    |   movel([0.307212, -1.318657, -2.613011, -0.780720, 1.570796, 1.878009],accel_mss,speed_ms,0,blend_radius_m)
    |   movel([0.307312, -1.318721, -2.612972, -0.780696, 1.570796, 1.878109],accel_mss,speed_ms,0,blend_radius_m)
    |   movel([0.307553, -1.318455, -2.613136, -0.780797, 1.570796, 1.878349],accel_mss,speed_ms,0,blend_radius_m)
    |   movel([0.309131, -1.316503, -2.614344, -0.781542, 1.570796, 1.879927],accel_mss,speed_ms,0,blend_radius_m)
    |   movel([0.310529, -1.314958, -2.615295, -0.782136, 1.570796, 1.881325],accel_mss,speed_ms,0,blend_radius_m)
    |   movel([0.313319, -1.312233, -2.616967, -0.783190, 1.570796, 1.884115],accel_mss,speed_ms,0,blend_radius_m)
    |   movel([0.314719, -1.311087, -2.617666, -0.783636, 1.570796, 1.885515],accel_mss,speed_ms,0,blend_radius_m)
    |   movel([0.316170, -1.310050, -2.618298, -0.784041, 1.570796, 1.886966],accel_mss,speed_ms,0,blend_radius_m)
    |   movel([0.317768, -1.309055, -2.618903, -0.784431, 1.570796, 1.888565],accel_mss,speed_ms,0,blend_radius_m)
    |   movel([0.321234, -1.307125, -2.620073, -0.785192, 1.570796, 1.892031],accel_mss,speed_ms,0,blend_radius_m)
    |   movel([0.322560, -1.306227, -2.620615, -0.785547, 1.570796, 1.893356],accel_mss,speed_ms,0,blend_radius_m)
    |   movel([0.323660, -1.305298, -2.621175, -0.785916, 1.570796, 1.894456],accel_mss,speed_ms,0,blend_radius_m)
    |   movel([0.324594, -1.304294, -2.621779, -0.786316, 1.570796, 1.895391],accel_mss,speed_ms,0,blend_radius_m)
    |   movel([0.325732, -1.302493, -2.622860, -0.787037, 1.570796, 1.896528],accel_mss,speed_ms,0,blend_radius_m)
    |   movel([0.326232, -1.301501, -2.623453, -0.787435, 1.570796, 1.897028],accel_mss,speed_ms,0,blend_radius_m)
    |   movel([0.326144, -1.301362, -2.623536, -0.787491, 1.570796, 1.896941],accel_mss,speed_ms,0,blend_radius_m)
    |   movel([0.325589, -1.301882, -2.623225, -0.787282, 1.570796, 1.896385],accel_mss,speed_ms,0,blend_radius_m)
    |   movel([0.325038, -1.302447, -2.622887, -0.787055, 1.570796, 1.895835],accel_mss,speed_ms,0,blend_radius_m)
    |   movel([0.323893, -1.303624, -2.622182, -0.786584, 1.570796, 1.894689],accel_mss,speed_ms,0,blend_radius_m)
    |   speed_ms = 0.005
    |   movel([0.323893, -1.294431, -2.617839, -0.800119, 1.570796, 1.894689],accel_mss,speed_ms,0,blend_radius_m)
    |   speed_ms = 0.040
    |   movel([0.326258, -1.294277, -2.617930, -0.800182, 1.570796, 1.897054],accel_mss,speed_ms,0,blend_radius_m)
    |   speed_ms = 0.005
    |   movel([0.326258, -1.303470, -2.622274, -0.786645, 1.570796, 1.897054],accel_mss,speed_ms,0,blend_radius_m)
    |   speed_ms = 0.025
    |   movel([0.326747, -1.302560, -2.622819, -0.787009, 1.570796, 1.897543],accel_mss,speed_ms,0,blend_radius_m)
    |   movel([0.327247, -1.301359, -2.623537, -0.787492, 1.570796, 1.898043],accel_mss,speed_ms,0,blend_radius_m)
    |   movel([0.327645, -1.300186, -2.624237, -0.787966, 1.570796, 1.898441],accel_mss,speed_ms,0,blend_radius_m)
    |   movel([0.327795, -1.299396, -2.624707, -0.788286, 1.570796, 1.898591],accel_mss,speed_ms,0,blend_radius_m)
    |   movel([0.327707, -1.299045, -2.624916, -0.788428, 1.570796, 1.898503],accel_mss,speed_ms,0,blend_radius_m)
    |   movel([0.327425, -1.298928, -2.624985, -0.788475, 1.570796, 1.898222],accel_mss,speed_ms,0,blend_radius_m)
    |   movel([0.327033, -1.299087, -2.624891, -0.788411, 1.570796, 1.897830],accel_mss,speed_ms,0,blend_radius_m)
    |   movel([0.326013, -1.300232, -2.624210, -0.787947, 1.570796, 1.896809],accel_mss,speed_ms,0,blend_radius_m)
    |   movel([0.325507, -1.300775, -2.623886, -0.787728, 1.570796, 1.896303],accel_mss,speed_ms,0,blend_radius_m)
    |   movel([0.321787, -1.304518, -2.621645, -0.786227, 1.570796, 1.892583],accel_mss,speed_ms,0,blend_radius_m)
    |   movel([0.320328, -1.305732, -2.620914, -0.785744, 1.570796, 1.891125],accel_mss,speed_ms,0,blend_radius_m)
    |   movel([0.315897, -1.308955, -2.618964, -0.784470, 1.570796, 1.886693],accel_mss,speed_ms,0,blend_radius_m)
    |   movel([0.313137, -1.310933, -2.617760, -0.783696, 1.570796, 1.883934],accel_mss,speed_ms,0,blend_radius_m)
    |   movel([0.311061, -1.312571, -2.616760, -0.783058, 1.570796, 1.881857],accel_mss,speed_ms,0,blend_radius_m)
    |   movel([0.309487, -1.314003, -2.615882, -0.782504, 1.570796, 1.880283],accel_mss,speed_ms,0,blend_radius_m)
    |   movel([0.308299, -1.315334, -2.615064, -0.781991, 1.570796, 1.879095],accel_mss,speed_ms,0,blend_radius_m)
    |   movel([0.306934, -1.317318, -2.613840, -0.781231, 1.570796, 1.877730],accel_mss,speed_ms,0,blend_radius_m)
    |   movel([0.306002, -1.319214, -2.612666, -0.780509, 1.570796, 1.876798],accel_mss,speed_ms,0,blend_radius_m)
    |   movel([0.305550, -1.320906, -2.611614, -0.779869, 1.570796, 1.876346],accel_mss,speed_ms,0,blend_radius_m)
    |   movel([0.305606, -1.322295, -2.610747, -0.779347, 1.570796, 1.876402],accel_mss,speed_ms,0,blend_radius_m)
    |   movel([0.305810, -1.322929, -2.610351, -0.779109, 1.570796, 1.876606],accel_mss,speed_ms,0,blend_radius_m)
    |   movel([0.306043, -1.323253, -2.610148, -0.778988, 1.570796, 1.876840],accel_mss,speed_ms,0,blend_radius_m)
    |   movel([0.306324, -1.323321, -2.610106, -0.778962, 1.570796, 1.877120],accel_mss,speed_ms,0,blend_radius_m)
    |   movel([0.306667, -1.323175, -2.610197, -0.779017, 1.570796, 1.877463],accel_mss,speed_ms,0,blend_radius_m)
    |   movel([0.306853, -1.323006, -2.610303, -0.779080, 1.570796, 1.877649],accel_mss,speed_ms,0,blend_radius_m)
    |   movel([0.306996, -1.322598, -2.610558, -0.779233, 1.570796, 1.877793],accel_mss,speed_ms,0,blend_radius_m)
    |   movel([0.306995, -1.322152, -2.610837, -0.779400, 1.570796, 1.877792],accel_mss,speed_ms,0,blend_radius_m)
    |   movel([0.307215, -1.320929, -2.611600, -0.779861, 1.570796, 1.878011],accel_mss,speed_ms,0,blend_radius_m)
    |   movel([0.307915, -1.319503, -2.612487, -0.780400, 1.570796, 1.878712],accel_mss,speed_ms,0,blend_radius_m)
    |   movel([0.309145, -1.317798, -2.613544, -0.781048, 1.570796, 1.879941],accel_mss,speed_ms,0,blend_radius_m)
    |   movel([0.310979, -1.315725, -2.614823, -0.781841, 1.570796, 1.881775],accel_mss,speed_ms,0,blend_radius_m)
    |   movel([0.313038, -1.313657, -2.616095, -0.782638, 1.570796, 1.883835],accel_mss,speed_ms,0,blend_radius_m)
    |   movel([0.314866, -1.312075, -2.617063, -0.783251, 1.570796, 1.885662],accel_mss,speed_ms,0,blend_radius_m)
    |   movel([0.316790, -1.310710, -2.617896, -0.783783, 1.570796, 1.887586],accel_mss,speed_ms,0,blend_radius_m)
    |   movel([0.319152, -1.309304, -2.618752, -0.784333, 1.570796, 1.889949],accel_mss,speed_ms,0,blend_radius_m)
    |   movel([0.322628, -1.307240, -2.620003, -0.785146, 1.570796, 1.893424],accel_mss,speed_ms,0,blend_radius_m)
    |   movel([0.323637, -1.306466, -2.620471, -0.785452, 1.570796, 1.894434],accel_mss,speed_ms,0,blend_radius_m)
    |   movel([0.324629, -1.305529, -2.621036, -0.785824, 1.570796, 1.895425],accel_mss,speed_ms,0,blend_radius_m)
    |   movel([0.325525, -1.304506, -2.621652, -0.786231, 1.570796, 1.896322],accel_mss,speed_ms,0,blend_radius_m)
    |   movel([0.326258, -1.303470, -2.622274, -0.786645, 1.570796, 1.897054],accel_mss,speed_ms,0,blend_radius_m)
    |   movel([0.326747, -1.302560, -2.622819, -0.787009, 1.570796, 1.897543],accel_mss,speed_ms,0,blend_radius_m)
    |   movel([0.327247, -1.301359, -2.623537, -0.787492, 1.570796, 1.898043],accel_mss,speed_ms,0,blend_radius_m)
    |   movel([0.327406, -1.300891, -2.623817, -0.787681, 1.570796, 1.898202],accel_mss,speed_ms,0,blend_radius_m)
    |   speed_ms = 0.005
    |   movel([0.327406, -1.291683, -2.619461, -0.801245, 1.570796, 1.898202],accel_mss,speed_ms,0,blend_radius_m)
    |   speed_ms = 0.040
    |   movel([0.337782, -1.301882, -2.613390, -0.797116, 1.570796, 1.908579],accel_mss,speed_ms,0,blend_radius_m)
    |   speed_ms = 0.005
    |   movel([0.337782, -1.311032, -2.617700, -0.783657, 1.570796, 1.908579],accel_mss,speed_ms,0,blend_radius_m)
    |   speed_ms = 0.025
    |   movel([0.338243, -1.310133, -2.618248, -0.784008, 1.570796, 1.909039],accel_mss,speed_ms,0,blend_radius_m)
    |   movel([0.339898, -1.306587, -2.620397, -0.785404, 1.570796, 1.910694],accel_mss,speed_ms,0,blend_radius_m)
    |   movel([0.340033, -1.306182, -2.620642, -0.785565, 1.570796, 1.910829],accel_mss,speed_ms,0,blend_radius_m)
    |   movel([0.339919, -1.305852, -2.620841, -0.785696, 1.570796, 1.910716],accel_mss,speed_ms,0,blend_radius_m)
    |   movel([0.339552, -1.305923, -2.620798, -0.785668, 1.570796, 1.910349],accel_mss,speed_ms,0,blend_radius_m)
    |   movel([0.339171, -1.306264, -2.620593, -0.785533, 1.570796, 1.909967],accel_mss,speed_ms,0,blend_radius_m)
    |   movel([0.338711, -1.306998, -2.620149, -0.785242, 1.570796, 1.909508],accel_mss,speed_ms,0,blend_radius_m)
    |   movel([0.336280, -1.311905, -2.617167, -0.783317, 1.570796, 1.907076],accel_mss,speed_ms,0,blend_radius_m)
    |   movel([0.335256, -1.313851, -2.615976, -0.782563, 1.570796, 1.906053],accel_mss,speed_ms,0,blend_radius_m)
    |   movel([0.335041, -1.314109, -2.615817, -0.782463, 1.570796, 1.905837],accel_mss,speed_ms,0,blend_radius_m)
    |   movel([0.333925, -1.313709, -2.616063, -0.782617, 1.570796, 1.904721],accel_mss,speed_ms,0,blend_radius_m)
    |   movel([0.333466, -1.313809, -2.616001, -0.782579, 1.570796, 1.904262],accel_mss,speed_ms,0,blend_radius_m)
    |   movel([0.332950, -1.314205, -2.615758, -0.782426, 1.570796, 1.903746],accel_mss,speed_ms,0,blend_radius_m)
    |   movel([0.332250, -1.315025, -2.615254, -0.782110, 1.570796, 1.903046],accel_mss,speed_ms,0,blend_radius_m)
    |   movel([0.330578, -1.316890, -2.614105, -0.781394, 1.570796, 1.901374],accel_mss,speed_ms,0,blend_radius_m)
    |   movel([0.329691, -1.317759, -2.613568, -0.781062, 1.570796, 1.900487],accel_mss,speed_ms,0,blend_radius_m)
    |   movel([0.329694, -1.317312, -2.613844, -0.781233, 1.570796, 1.900490],accel_mss,speed_ms,0,blend_radius_m)
    |   movel([0.329719, -1.317037, -2.614014, -0.781338, 1.570796, 1.900515],accel_mss,speed_ms,0,blend_radius_m)
    |   movel([0.330422, -1.313511, -2.616184, -0.782694, 1.570796, 1.901218],accel_mss,speed_ms,0,blend_radius_m)
    |   movel([0.330386, -1.313253, -2.616342, -0.782794, 1.570796, 1.901182],accel_mss,speed_ms,0,blend_radius_m)
    |   movel([0.330238, -1.313153, -2.616403, -0.782833, 1.570796, 1.901034],accel_mss,speed_ms,0,blend_radius_m)
    |   movel([0.330096, -1.313161, -2.616398, -0.782829, 1.570796, 1.900892],accel_mss,speed_ms,0,blend_radius_m)
    |   movel([0.329664, -1.313389, -2.616259, -0.782741, 1.570796, 1.900460],accel_mss,speed_ms,0,blend_radius_m)
    |   movel([0.329304, -1.314002, -2.615883, -0.782504, 1.570796, 1.900100],accel_mss,speed_ms,0,blend_radius_m)
    |   movel([0.328587, -1.317415, -2.613780, -0.781194, 1.570796, 1.899383],accel_mss,speed_ms,0,blend_radius_m)
    |   movel([0.328597, -1.318361, -2.613195, -0.780833, 1.570796, 1.899393],accel_mss,speed_ms,0,blend_radius_m)
    |   movel([0.328770, -1.318650, -2.613016, -0.780723, 1.570796, 1.899566],accel_mss,speed_ms,0,blend_radius_m)
    |   movel([0.329121, -1.318773, -2.612940, -0.780677, 1.570796, 1.899918],accel_mss,speed_ms,0,blend_radius_m)
    |   movel([0.329584, -1.318705, -2.612981, -0.780702, 1.570796, 1.900380],accel_mss,speed_ms,0,blend_radius_m)
    |   movel([0.330062, -1.318458, -2.613135, -0.780796, 1.570796, 1.900859],accel_mss,speed_ms,0,blend_radius_m)
    |   movel([0.330544, -1.318068, -2.613376, -0.780944, 1.570796, 1.901341],accel_mss,speed_ms,0,blend_radius_m)
    |   movel([0.331223, -1.317416, -2.613780, -0.781193, 1.570796, 1.902019],accel_mss,speed_ms,0,blend_radius_m)
    |   movel([0.333567, -1.314812, -2.615385, -0.782192, 1.570796, 1.904363],accel_mss,speed_ms,0,blend_radius_m)
    |   movel([0.334016, -1.315298, -2.615086, -0.782005, 1.570796, 1.904812],accel_mss,speed_ms,0,blend_radius_m)
    |   movel([0.334664, -1.315728, -2.614822, -0.781840, 1.570796, 1.905460],accel_mss,speed_ms,0,blend_radius_m)
    |   movel([0.334838, -1.315746, -2.614811, -0.781833, 1.570796, 1.905634],accel_mss,speed_ms,0,blend_radius_m)
    |   movel([0.335212, -1.315522, -2.614948, -0.781919, 1.570796, 1.906008],accel_mss,speed_ms,0,blend_radius_m)
    |   movel([0.335737, -1.314781, -2.615404, -0.782204, 1.570796, 1.906534],accel_mss,speed_ms,0,blend_radius_m)
    |   movel([0.337782, -1.311032, -2.617700, -0.783657, 1.570796, 1.908579],accel_mss,speed_ms,0,blend_radius_m)
    |   movel([0.338243, -1.310133, -2.618248, -0.784008, 1.570796, 1.909039],accel_mss,speed_ms,0,blend_radius_m)
    |   movel([0.339015, -1.308475, -2.619255, -0.784659, 1.570796, 1.909811],accel_mss,speed_ms,0,blend_radius_m)
    |   speed_ms = 0.005
    |   movel([0.339015, -1.299311, -2.614934, -0.798145, 1.570796, 1.909811],accel_mss,speed_ms,0,blend_radius_m)
    |   speed_ms = 0.040
    |   movel([0.312088, -1.325803, -2.598622, -0.787964, 1.570796, 1.882884],accel_mss,speed_ms,0,blend_radius_m)
    |   speed_ms = 0.005
    |   movel([0.312088, -1.334807, -2.602825, -0.774757, 1.570796, 1.882884],accel_mss,speed_ms,0,blend_radius_m)
    |   speed_ms = 0.025
    |   movel([0.308392, -1.337491, -2.601098, -0.773800, 1.570796, 1.879188],accel_mss,speed_ms,0,blend_radius_m)
    |   movel([0.307353, -1.338080, -2.600717, -0.773591, 1.570796, 1.878150],accel_mss,speed_ms,0,blend_radius_m)
    |   movel([0.306493, -1.338398, -2.600512, -0.773479, 1.570796, 1.877289],accel_mss,speed_ms,0,blend_radius_m)
    |   movel([0.305914, -1.338470, -2.600466, -0.773453, 1.570796, 1.876710],accel_mss,speed_ms,0,blend_radius_m)
    |   movel([0.305711, -1.338314, -2.600567, -0.773509, 1.570796, 1.876508],accel_mss,speed_ms,0,blend_radius_m)
    |   movel([0.305836, -1.337950, -2.600802, -0.773637, 1.570796, 1.876632],accel_mss,speed_ms,0,blend_radius_m)
    |   movel([0.308276, -1.335053, -2.602667, -0.774669, 1.570796, 1.879072],accel_mss,speed_ms,0,blend_radius_m)
    |   movel([0.309248, -1.333743, -2.603507, -0.775139, 1.570796, 1.880044],accel_mss,speed_ms,0,blend_radius_m)
    |   movel([0.310608, -1.331652, -2.604842, -0.775894, 1.570796, 1.881405],accel_mss,speed_ms,0,blend_radius_m)
    |   movel([0.310997, -1.330924, -2.605306, -0.776159, 1.570796, 1.881794],accel_mss,speed_ms,0,blend_radius_m)
    |   movel([0.312034, -1.328173, -2.607052, -0.777164, 1.570796, 1.882830],accel_mss,speed_ms,0,blend_radius_m)
    |   movel([0.312141, -1.327720, -2.607338, -0.777331, 1.570796, 1.882937],accel_mss,speed_ms,0,blend_radius_m)
    |   movel([0.311958, -1.327277, -2.607618, -0.777494, 1.570796, 1.882755],accel_mss,speed_ms,0,blend_radius_m)
    |   movel([0.311748, -1.327028, -2.607775, -0.777586, 1.570796, 1.882544],accel_mss,speed_ms,0,blend_radius_m)
    |   movel([0.311758, -1.326727, -2.607965, -0.777697, 1.570796, 1.882554],accel_mss,speed_ms,0,blend_radius_m)
    |   movel([0.311983, -1.326441, -2.608145, -0.777802, 1.570796, 1.882779],accel_mss,speed_ms,0,blend_radius_m)
    |   movel([0.312368, -1.326236, -2.608275, -0.777878, 1.570796, 1.883164],accel_mss,speed_ms,0,blend_radius_m)
    |   movel([0.312840, -1.326193, -2.608302, -0.777894, 1.570796, 1.883637],accel_mss,speed_ms,0,blend_radius_m)
    |   movel([0.313138, -1.326410, -2.608165, -0.777814, 1.570796, 1.883934],accel_mss,speed_ms,0,blend_radius_m)
    |   movel([0.313250, -1.326915, -2.607847, -0.777627, 1.570796, 1.884046],accel_mss,speed_ms,0,blend_radius_m)
    |   movel([0.313171, -1.327736, -2.607328, -0.777325, 1.570796, 1.883967],accel_mss,speed_ms,0,blend_radius_m)
    |   movel([0.312702, -1.329366, -2.606296, -0.776727, 1.570796, 1.883499],accel_mss,speed_ms,0,blend_radius_m)
    |   movel([0.311799, -1.331308, -2.605062, -0.776019, 1.570796, 1.882595],accel_mss,speed_ms,0,blend_radius_m)
    |   movel([0.310569, -1.333362, -2.603751, -0.775276, 1.570796, 1.881366],accel_mss,speed_ms,0,blend_radius_m)
    |   movel([0.308247, -1.336526, -2.601720, -0.774143, 1.570796, 1.879043],accel_mss,speed_ms,0,blend_radius_m)
    |   movel([0.309250, -1.335888, -2.602131, -0.774370, 1.570796, 1.880046],accel_mss,speed_ms,0,blend_radius_m)
    |   movel([0.310249, -1.335148, -2.602606, -0.774635, 1.570796, 1.881045],accel_mss,speed_ms,0,blend_radius_m)
    |   movel([0.313227, -1.332919, -2.604034, -0.775436, 1.570796, 1.884024],accel_mss,speed_ms,0,blend_radius_m)
    |   movel([0.314209, -1.332259, -2.604455, -0.775674, 1.570796, 1.885005],accel_mss,speed_ms,0,blend_radius_m)
    |   movel([0.314787, -1.331983, -2.604632, -0.775775, 1.570796, 1.885583],accel_mss,speed_ms,0,blend_radius_m)
    |   movel([0.315091, -1.332027, -2.604603, -0.775758, 1.570796, 1.885887],accel_mss,speed_ms,0,blend_radius_m)
    |   movel([0.315060, -1.332306, -2.604426, -0.775658, 1.570796, 1.885856],accel_mss,speed_ms,0,blend_radius_m)
    |   movel([0.314691, -1.332734, -2.604152, -0.775503, 1.570796, 1.885488],accel_mss,speed_ms,0,blend_radius_m)
    |   movel([0.312088, -1.334807, -2.602825, -0.774757, 1.570796, 1.882884],accel_mss,speed_ms,0,blend_radius_m)
    |   movel([0.309627, -1.336591, -2.601678, -0.774120, 1.570796, 1.880423],accel_mss,speed_ms,0,blend_radius_m)
    |   speed_ms = 0.005
    |   movel([0.309627, -1.327599, -2.597483, -0.787307, 1.570796, 1.880423],accel_mss,speed_ms,0,blend_radius_m)
    |   speed_ms = 0.040
    |   movel([0.307273, -1.324388, -2.599517, -0.788484, 1.570796, 1.878069],accel_mss,speed_ms,0,blend_radius_m)
    |   speed_ms = 0.005
    |   movel([0.307273, -1.333401, -2.603726, -0.775262, 1.570796, 1.878069],accel_mss,speed_ms,0,blend_radius_m)
    |   speed_ms = 0.025
    |   movel([0.308595, -1.332314, -2.604420, -0.775655, 1.570796, 1.879391],accel_mss,speed_ms,0,blend_radius_m)
    |   movel([0.309287, -1.331629, -2.604857, -0.775903, 1.570796, 1.880084],accel_mss,speed_ms,0,blend_radius_m)
    |   movel([0.309505, -1.331215, -2.605121, -0.776053, 1.570796, 1.880302],accel_mss,speed_ms,0,blend_radius_m)
    |   movel([0.309377, -1.330977, -2.605272, -0.776139, 1.570796, 1.880173],accel_mss,speed_ms,0,blend_radius_m)
    |   movel([0.309182, -1.331020, -2.605245, -0.776124, 1.570796, 1.879979],accel_mss,speed_ms,0,blend_radius_m)
    |   movel([0.308663, -1.331351, -2.605035, -0.776004, 1.570796, 1.879459],accel_mss,speed_ms,0,blend_radius_m)
    |   movel([0.304437, -1.334482, -2.603033, -0.774873, 1.570796, 1.875234],accel_mss,speed_ms,0,blend_radius_m)
    |   movel([0.301937, -1.336094, -2.601998, -0.774297, 1.570796, 1.872734],accel_mss,speed_ms,0,blend_radius_m)
    |   movel([0.299591, -1.337354, -2.601187, -0.773849, 1.570796, 1.870388],accel_mss,speed_ms,0,blend_radius_m)
    |   movel([0.297404, -1.338260, -2.600601, -0.773528, 1.570796, 1.868201],accel_mss,speed_ms,0,blend_radius_m)
    |   movel([0.295735, -1.338801, -2.600251, -0.773336, 1.570796, 1.866531],accel_mss,speed_ms,0,blend_radius_m)
    |   movel([0.298270, -1.336381, -2.601813, -0.774195, 1.570796, 1.869067],accel_mss,speed_ms,0,blend_radius_m)
    |   movel([0.299778, -1.334767, -2.602851, -0.774771, 1.570796, 1.870574],accel_mss,speed_ms,0,blend_radius_m)
    |   movel([0.301019, -1.333262, -2.603815, -0.775312, 1.570796, 1.871816],accel_mss,speed_ms,0,blend_radius_m)
    |   movel([0.301505, -1.332372, -2.604383, -0.775634, 1.570796, 1.872302],accel_mss,speed_ms,0,blend_radius_m)
    |   movel([0.301499, -1.332129, -2.604538, -0.775721, 1.570796, 1.872295],accel_mss,speed_ms,0,blend_radius_m)
    |   movel([0.301389, -1.332106, -2.604553, -0.775730, 1.570796, 1.872185],accel_mss,speed_ms,0,blend_radius_m)
    |   movel([0.300923, -1.332271, -2.604448, -0.775670, 1.570796, 1.871719],accel_mss,speed_ms,0,blend_radius_m)
    |   movel([0.300572, -1.332571, -2.604256, -0.775562, 1.570796, 1.871369],accel_mss,speed_ms,0,blend_radius_m)
    |   movel([0.299480, -1.333796, -2.603473, -0.775120, 1.570796, 1.870276],accel_mss,speed_ms,0,blend_radius_m)
    |   movel([0.298256, -1.335199, -2.602573, -0.774617, 1.570796, 1.869053],accel_mss,speed_ms,0,blend_radius_m)
    |   movel([0.297100, -1.336370, -2.601820, -0.774198, 1.570796, 1.867896],accel_mss,speed_ms,0,blend_radius_m)
    |   movel([0.295923, -1.337399, -2.601157, -0.773833, 1.570796, 1.866720],accel_mss,speed_ms,0,blend_radius_m)
    |   movel([0.293513, -1.339225, -2.599977, -0.773187, 1.570796, 1.864309],accel_mss,speed_ms,0,blend_radius_m)
    |   movel([0.293230, -1.339512, -2.599791, -0.773086, 1.570796, 1.864027],accel_mss,speed_ms,0,blend_radius_m)
    |   movel([0.293138, -1.339896, -2.599542, -0.772951, 1.570796, 1.863934],accel_mss,speed_ms,0,blend_radius_m)
    |   movel([0.293264, -1.339985, -2.599484, -0.772920, 1.570796, 1.864061],accel_mss,speed_ms,0,blend_radius_m)
    |   movel([0.294226, -1.339955, -2.599504, -0.772930, 1.570796, 1.865022],accel_mss,speed_ms,0,blend_radius_m)
    |   movel([0.295597, -1.339742, -2.599642, -0.773005, 1.570796, 1.866393],accel_mss,speed_ms,0,blend_radius_m)
    |   movel([0.297004, -1.339349, -2.599897, -0.773143, 1.570796, 1.867801],accel_mss,speed_ms,0,blend_radius_m)
    |   movel([0.298619, -1.338737, -2.600293, -0.773359, 1.570796, 1.869415],accel_mss,speed_ms,0,blend_radius_m)
    |   movel([0.300228, -1.337994, -2.600773, -0.773622, 1.570796, 1.871025],accel_mss,speed_ms,0,blend_radius_m)
    |   movel([0.301988, -1.337043, -2.601387, -0.773959, 1.570796, 1.872784],accel_mss,speed_ms,0,blend_radius_m)
    |   movel([0.303714, -1.335978, -2.602073, -0.774338, 1.570796, 1.874511],accel_mss,speed_ms,0,blend_radius_m)
    |   movel([0.305518, -1.334733, -2.602872, -0.774783, 1.570796, 1.876314],accel_mss,speed_ms,0,blend_radius_m)
    |   movel([0.307273, -1.333401, -2.603726, -0.775262, 1.570796, 1.878069],accel_mss,speed_ms,0,blend_radius_m)
    |   movel([0.308595, -1.332314, -2.604420, -0.775655, 1.570796, 1.879391],accel_mss,speed_ms,0,blend_radius_m)
    |   movel([0.309287, -1.331629, -2.604857, -0.775903, 1.570796, 1.880084],accel_mss,speed_ms,0,blend_radius_m)
    |   movel([0.309446, -1.331328, -2.605049, -0.776012, 1.570796, 1.880242],accel_mss,speed_ms,0,blend_radius_m)
    |   speed_ms = 0.005
    |   movel([0.309446, -1.322303, -2.600830, -0.789256, 1.570796, 1.880242],accel_mss,speed_ms,0,blend_radius_m)
    |   speed_ms = 0.040
    |   movel([0.281169, -1.327397, -2.597611, -0.787380, 1.570796, 1.851966],accel_mss,speed_ms,0,blend_radius_m)
    |   speed_ms = 0.005
    |   movel([0.281169, -1.336390, -2.601807, -0.774191, 1.570796, 1.851966],accel_mss,speed_ms,0,blend_radius_m)
    |   speed_ms = 0.025
    |   movel([0.281589, -1.336173, -2.601948, -0.774269, 1.570796, 1.852385],accel_mss,speed_ms,0,blend_radius_m)
    |   movel([0.281862, -1.335916, -2.602113, -0.774361, 1.570796, 1.852658],accel_mss,speed_ms,0,blend_radius_m)
    |   movel([0.281947, -1.335663, -2.602275, -0.774451, 1.570796, 1.852743],accel_mss,speed_ms,0,blend_radius_m)
    |   movel([0.281691, -1.335396, -2.602447, -0.774546, 1.570796, 1.852488],accel_mss,speed_ms,0,blend_radius_m)
    |   movel([0.281436, -1.335403, -2.602442, -0.774543, 1.570796, 1.852232],accel_mss,speed_ms,0,blend_radius_m)
    |   movel([0.280018, -1.335751, -2.602219, -0.774419, 1.570796, 1.850815],accel_mss,speed_ms,0,blend_radius_m)
    |   movel([0.279438, -1.335889, -2.602130, -0.774370, 1.570796, 1.850234],accel_mss,speed_ms,0,blend_radius_m)
    |   movel([0.277464, -1.336169, -2.601950, -0.774270, 1.570796, 1.848260],accel_mss,speed_ms,0,blend_radius_m)
    |   movel([0.276225, -1.336162, -2.601954, -0.774273, 1.570796, 1.847021],accel_mss,speed_ms,0,blend_radius_m)
    |   movel([0.274250, -1.335940, -2.602097, -0.774352, 1.570796, 1.845046],accel_mss,speed_ms,0,blend_radius_m)
    |   movel([0.273688, -1.335778, -2.602201, -0.774410, 1.570796, 1.844484],accel_mss,speed_ms,0,blend_radius_m)
    |   movel([0.274932, -1.335215, -2.602563, -0.774611, 1.570796, 1.845728],accel_mss,speed_ms,0,blend_radius_m)
    |   movel([0.276555, -1.334383, -2.603097, -0.774909, 1.570796, 1.847351],accel_mss,speed_ms,0,blend_radius_m)
    |   movel([0.278096, -1.333386, -2.603736, -0.775268, 1.570796, 1.848892],accel_mss,speed_ms,0,blend_radius_m)
    |   movel([0.279291, -1.332432, -2.604345, -0.775612, 1.570796, 1.850087],accel_mss,speed_ms,0,blend_radius_m)
    |   movel([0.279536, -1.332138, -2.604533, -0.775718, 1.570796, 1.850333],accel_mss,speed_ms,0,blend_radius_m)
    |   movel([0.279647, -1.331822, -2.604734, -0.775833, 1.570796, 1.850443],accel_mss,speed_ms,0,blend_radius_m)
    |   movel([0.279578, -1.331667, -2.604833, -0.775889, 1.570796, 1.850375],accel_mss,speed_ms,0,blend_radius_m)
    |   movel([0.279357, -1.331607, -2.604871, -0.775911, 1.570796, 1.850153],accel_mss,speed_ms,0,blend_radius_m)
    |   movel([0.277761, -1.331783, -2.604759, -0.775847, 1.570796, 1.848557],accel_mss,speed_ms,0,blend_radius_m)
    |   movel([0.275731, -1.331936, -2.604661, -0.775791, 1.570796, 1.846527],accel_mss,speed_ms,0,blend_radius_m)
    |   movel([0.274030, -1.331774, -2.604765, -0.775850, 1.570796, 1.844826],accel_mss,speed_ms,0,blend_radius_m)
    |   movel([0.272602, -1.331281, -2.605079, -0.776029, 1.570796, 1.843398],accel_mss,speed_ms,0,blend_radius_m)
    |   movel([0.271400, -1.330446, -2.605610, -0.776333, 1.570796, 1.842196],accel_mss,speed_ms,0,blend_radius_m)
    |   movel([0.270719, -1.329821, -2.606007, -0.776561, 1.570796, 1.841515],accel_mss,speed_ms,0,blend_radius_m)
    |   movel([0.272339, -1.329417, -2.606263, -0.776708, 1.570796, 1.843135],accel_mss,speed_ms,0,blend_radius_m)
    |   movel([0.273542, -1.328831, -2.606635, -0.776923, 1.570796, 1.844338],accel_mss,speed_ms,0,blend_radius_m)
    |   movel([0.274574, -1.328160, -2.607060, -0.777169, 1.570796, 1.845371],accel_mss,speed_ms,0,blend_radius_m)
    |   movel([0.274821, -1.327919, -2.607213, -0.777258, 1.570796, 1.845617],accel_mss,speed_ms,0,blend_radius_m)
    |   movel([0.274963, -1.327481, -2.607489, -0.777419, 1.570796, 1.845759],accel_mss,speed_ms,0,blend_radius_m)
    |   movel([0.274856, -1.327336, -2.607581, -0.777472, 1.570796, 1.845652],accel_mss,speed_ms,0,blend_radius_m)
    |   movel([0.273461, -1.326733, -2.607961, -0.777695, 1.570796, 1.844257],accel_mss,speed_ms,0,blend_radius_m)
    |   movel([0.272555, -1.326179, -2.608311, -0.777900, 1.570796, 1.843351],accel_mss,speed_ms,0,blend_radius_m)
    |   movel([0.270971, -1.324730, -2.609222, -0.778437, 1.570796, 1.841768],accel_mss,speed_ms,0,blend_radius_m)
    |   movel([0.270367, -1.323880, -2.609756, -0.778754, 1.570796, 1.841164],accel_mss,speed_ms,0,blend_radius_m)
    |   movel([0.268936, -1.321297, -2.611370, -0.779722, 1.570796, 1.839732],accel_mss,speed_ms,0,blend_radius_m)
    |   movel([0.269008, -1.321099, -2.611494, -0.779796, 1.570796, 1.839804],accel_mss,speed_ms,0,blend_radius_m)
    |   movel([0.269540, -1.321127, -2.611476, -0.779786, 1.570796, 1.840337],accel_mss,speed_ms,0,blend_radius_m)
    |   movel([0.270152, -1.321157, -2.611457, -0.779774, 1.570796, 1.840948],accel_mss,speed_ms,0,blend_radius_m)
    |   movel([0.271202, -1.321024, -2.611540, -0.779824, 1.570796, 1.841998],accel_mss,speed_ms,0,blend_radius_m)
    |   movel([0.272261, -1.320821, -2.611667, -0.779901, 1.570796, 1.843057],accel_mss,speed_ms,0,blend_radius_m)
    |   movel([0.272824, -1.320593, -2.611808, -0.779987, 1.570796, 1.843620],accel_mss,speed_ms,0,blend_radius_m)
    |   movel([0.272987, -1.320485, -2.611876, -0.780028, 1.570796, 1.843784],accel_mss,speed_ms,0,blend_radius_m)
    |   movel([0.273301, -1.320135, -2.612094, -0.780160, 1.570796, 1.844098],accel_mss,speed_ms,0,blend_radius_m)
    |   movel([0.273295, -1.319996, -2.612180, -0.780213, 1.570796, 1.844091],accel_mss,speed_ms,0,blend_radius_m)
    |   movel([0.270912, -1.316196, -2.614533, -0.781660, 1.570796, 1.841709],accel_mss,speed_ms,0,blend_radius_m)
    |   movel([0.270432, -1.315413, -2.615015, -0.781960, 1.570796, 1.841229],accel_mss,speed_ms,0,blend_radius_m)
    |   movel([0.269305, -1.313068, -2.616456, -0.782866, 1.570796, 1.840101],accel_mss,speed_ms,0,blend_radius_m)
    |   movel([0.268936, -1.312131, -2.617029, -0.783229, 1.570796, 1.839732],accel_mss,speed_ms,0,blend_radius_m)
    |   movel([0.268935, -1.311909, -2.617165, -0.783315, 1.570796, 1.839731],accel_mss,speed_ms,0,blend_radius_m)
    |   movel([0.271324, -1.312552, -2.616771, -0.783066, 1.570796, 1.842120],accel_mss,speed_ms,0,blend_radius_m)
    |   movel([0.271647, -1.312532, -2.616784, -0.783073, 1.570796, 1.842444],accel_mss,speed_ms,0,blend_radius_m)
    |   movel([0.271996, -1.312357, -2.616890, -0.783141, 1.570796, 1.842792],accel_mss,speed_ms,0,blend_radius_m)
    |   movel([0.272209, -1.312110, -2.617042, -0.783237, 1.570796, 1.843005],accel_mss,speed_ms,0,blend_radius_m)
    |   movel([0.272228, -1.311863, -2.617193, -0.783333, 1.570796, 1.843025],accel_mss,speed_ms,0,blend_radius_m)
    |   movel([0.271712, -1.310973, -2.617736, -0.783680, 1.570796, 1.842508],accel_mss,speed_ms,0,blend_radius_m)
    |   movel([0.270908, -1.309420, -2.618681, -0.784288, 1.570796, 1.841704],accel_mss,speed_ms,0,blend_radius_m)
    |   movel([0.270396, -1.307212, -2.620020, -0.785157, 1.570796, 1.841192],accel_mss,speed_ms,0,blend_radius_m)
    |   movel([0.270182, -1.304482, -2.621666, -0.786241, 1.570796, 1.840978],accel_mss,speed_ms,0,blend_radius_m)
    |   movel([0.270293, -1.301324, -2.623559, -0.787507, 1.570796, 1.841089],accel_mss,speed_ms,0,blend_radius_m)
    |   movel([0.270506, -1.299002, -2.624941, -0.788445, 1.570796, 1.841302],accel_mss,speed_ms,0,blend_radius_m)
    |   movel([0.271637, -1.300175, -2.624244, -0.787970, 1.570796, 1.842433],accel_mss,speed_ms,0,blend_radius_m)
    |   movel([0.272159, -1.300765, -2.623892, -0.787732, 1.570796, 1.842955],accel_mss,speed_ms,0,blend_radius_m)
    |   movel([0.272907, -1.301368, -2.623532, -0.787489, 1.570796, 1.843704],accel_mss,speed_ms,0,blend_radius_m)
    |   movel([0.273169, -1.301398, -2.623514, -0.787477, 1.570796, 1.843965],accel_mss,speed_ms,0,blend_radius_m)
    |   movel([0.273762, -1.301145, -2.623666, -0.787579, 1.570796, 1.844558],accel_mss,speed_ms,0,blend_radius_m)
    |   movel([0.273821, -1.301011, -2.623745, -0.787633, 1.570796, 1.844618],accel_mss,speed_ms,0,blend_radius_m)
    |   movel([0.273864, -1.299446, -2.624678, -0.788265, 1.570796, 1.844661],accel_mss,speed_ms,0,blend_radius_m)
    |   movel([0.273850, -1.298479, -2.625252, -0.788658, 1.570796, 1.844647],accel_mss,speed_ms,0,blend_radius_m)
    |   movel([0.273970, -1.291208, -2.629533, -0.791648, 1.570796, 1.844767],accel_mss,speed_ms,0,blend_radius_m)
    |   movel([0.274176, -1.287340, -2.631783, -0.793266, 1.570796, 1.844973],accel_mss,speed_ms,0,blend_radius_m)
    |   movel([0.274427, -1.286894, -2.632041, -0.793453, 1.570796, 1.845223],accel_mss,speed_ms,0,blend_radius_m)
    |   movel([0.275681, -1.288748, -2.630966, -0.792674, 1.570796, 1.846477],accel_mss,speed_ms,0,blend_radius_m)
    |   movel([0.276045, -1.289112, -2.630755, -0.792522, 1.570796, 1.846841],accel_mss,speed_ms,0,blend_radius_m)
    |   movel([0.276374, -1.289162, -2.630726, -0.792501, 1.570796, 1.847170],accel_mss,speed_ms,0,blend_radius_m)
    |   movel([0.276720, -1.288968, -2.630839, -0.792582, 1.570796, 1.847517],accel_mss,speed_ms,0,blend_radius_m)
    |   movel([0.276872, -1.288749, -2.630966, -0.792674, 1.570796, 1.847668],accel_mss,speed_ms,0,blend_radius_m)
    |   movel([0.276936, -1.288488, -2.631118, -0.792784, 1.570796, 1.847732],accel_mss,speed_ms,0,blend_radius_m)
    |   movel([0.276818, -1.287496, -2.631693, -0.793200, 1.570796, 1.847614],accel_mss,speed_ms,0,blend_radius_m)
    |   movel([0.276600, -1.285984, -2.632568, -0.793838, 1.570796, 1.847396],accel_mss,speed_ms,0,blend_radius_m)
    |   movel([0.276603, -1.284773, -2.633266, -0.794350, 1.570796, 1.847399],accel_mss,speed_ms,0,blend_radius_m)
    |   movel([0.276842, -1.283399, -2.634056, -0.794934, 1.570796, 1.847638],accel_mss,speed_ms,0,blend_radius_m)
    |   movel([0.278133, -1.279062, -2.636535, -0.796793, 1.570796, 1.848929],accel_mss,speed_ms,0,blend_radius_m)
    |   movel([0.278449, -1.278207, -2.637020, -0.797161, 1.570796, 1.849246],accel_mss,speed_ms,0,blend_radius_m)
    |   movel([0.278845, -1.277612, -2.637358, -0.797419, 1.570796, 1.849641],accel_mss,speed_ms,0,blend_radius_m)
    |   movel([0.279260, -1.278513, -2.636846, -0.797029, 1.570796, 1.850056],accel_mss,speed_ms,0,blend_radius_m)
    |   movel([0.279418, -1.279098, -2.636514, -0.796777, 1.570796, 1.850215],accel_mss,speed_ms,0,blend_radius_m)
    |   movel([0.279740, -1.279576, -2.636242, -0.796571, 1.570796, 1.850536],accel_mss,speed_ms,0,blend_radius_m)
    |   movel([0.279962, -1.279602, -2.636227, -0.796560, 1.570796, 1.850758],accel_mss,speed_ms,0,blend_radius_m)
    |   movel([0.280323, -1.279456, -2.636311, -0.796623, 1.570796, 1.851120],accel_mss,speed_ms,0,blend_radius_m)
    |   movel([0.280542, -1.279207, -2.636452, -0.796730, 1.570796, 1.851338],accel_mss,speed_ms,0,blend_radius_m)
    |   movel([0.280712, -1.277787, -2.637259, -0.797343, 1.570796, 1.851509],accel_mss,speed_ms,0,blend_radius_m)
    |   movel([0.280895, -1.276342, -2.638077, -0.797970, 1.570796, 1.851691],accel_mss,speed_ms,0,blend_radius_m)
    |   movel([0.281383, -1.274385, -2.639181, -0.798823, 1.570796, 1.852179],accel_mss,speed_ms,0,blend_radius_m)
    |   movel([0.282040, -1.272367, -2.640314, -0.799708, 1.570796, 1.852836],accel_mss,speed_ms,0,blend_radius_m)
    |   movel([0.283334, -1.269598, -2.641862, -0.800930, 1.570796, 1.854130],accel_mss,speed_ms,0,blend_radius_m)
    |   movel([0.284030, -1.268377, -2.642540, -0.801471, 1.570796, 1.854826],accel_mss,speed_ms,0,blend_radius_m)
    |   movel([0.285181, -1.266600, -2.643526, -0.802263, 1.570796, 1.855978],accel_mss,speed_ms,0,blend_radius_m)
    |   movel([0.278484, -1.290136, -2.630158, -0.792094, 1.570796, 1.849281],accel_mss,speed_ms,0,blend_radius_m)
    |   movel([0.276921, -1.295658, -2.626921, -0.789810, 1.570796, 1.847717],accel_mss,speed_ms,0,blend_radius_m)
    |   movel([0.275389, -1.301455, -2.623480, -0.787454, 1.570796, 1.846185],accel_mss,speed_ms,0,blend_radius_m)
    |   movel([0.274554, -1.306620, -2.620377, -0.785391, 1.570796, 1.845351],accel_mss,speed_ms,0,blend_radius_m)
    |   movel([0.274120, -1.311508, -2.617409, -0.783471, 1.570796, 1.844916],accel_mss,speed_ms,0,blend_radius_m)
    |   movel([0.274094, -1.315860, -2.614740, -0.781789, 1.570796, 1.844890],accel_mss,speed_ms,0,blend_radius_m)
    |   movel([0.274490, -1.319404, -2.612548, -0.780437, 1.570796, 1.845286],accel_mss,speed_ms,0,blend_radius_m)
    |   movel([0.274833, -1.320766, -2.611701, -0.779922, 1.570796, 1.845630],accel_mss,speed_ms,0,blend_radius_m)
    |   movel([0.275323, -1.322040, -2.610907, -0.779442, 1.570796, 1.846119],accel_mss,speed_ms,0,blend_radius_m)
    |   movel([0.275945, -1.323183, -2.610192, -0.779014, 1.570796, 1.846741],accel_mss,speed_ms,0,blend_radius_m)
    |   movel([0.276713, -1.324213, -2.609547, -0.778630, 1.570796, 1.847509],accel_mss,speed_ms,0,blend_radius_m)
    |   movel([0.277660, -1.325170, -2.608946, -0.778273, 1.570796, 1.848457],accel_mss,speed_ms,0,blend_radius_m)
    |   movel([0.278736, -1.326004, -2.608421, -0.777964, 1.570796, 1.849532],accel_mss,speed_ms,0,blend_radius_m)
    |   movel([0.280052, -1.326810, -2.607913, -0.777666, 1.570796, 1.850848],accel_mss,speed_ms,0,blend_radius_m)
    |   movel([0.282073, -1.327768, -2.607308, -0.777313, 1.570796, 1.852870],accel_mss,speed_ms,0,blend_radius_m)
    |   movel([0.282343, -1.327826, -2.607271, -0.777292, 1.570796, 1.853139],accel_mss,speed_ms,0,blend_radius_m)
    |   movel([0.282844, -1.327570, -2.607433, -0.777386, 1.570796, 1.853640],accel_mss,speed_ms,0,blend_radius_m)
    |   movel([0.283094, -1.327338, -2.607579, -0.777471, 1.570796, 1.853890],accel_mss,speed_ms,0,blend_radius_m)
    |   movel([0.283122, -1.327095, -2.607733, -0.777561, 1.570796, 1.853918],accel_mss,speed_ms,0,blend_radius_m)
    |   movel([0.282896, -1.326892, -2.607861, -0.777636, 1.570796, 1.853692],accel_mss,speed_ms,0,blend_radius_m)
    |   movel([0.281185, -1.325946, -2.608457, -0.777986, 1.570796, 1.851981],accel_mss,speed_ms,0,blend_radius_m)
    |   movel([0.279868, -1.325215, -2.608917, -0.778257, 1.570796, 1.850665],accel_mss,speed_ms,0,blend_radius_m)
    |   movel([0.278657, -1.324324, -2.609477, -0.778588, 1.570796, 1.849453],accel_mss,speed_ms,0,blend_radius_m)
    |   movel([0.277641, -1.323357, -2.610083, -0.778949, 1.570796, 1.848437],accel_mss,speed_ms,0,blend_radius_m)
    |   movel([0.276926, -1.322389, -2.610688, -0.779311, 1.570796, 1.847722],accel_mss,speed_ms,0,blend_radius_m)
    |   movel([0.276395, -1.321223, -2.611416, -0.779750, 1.570796, 1.847191],accel_mss,speed_ms,0,blend_radius_m)
    |   movel([0.275478, -1.317626, -2.613650, -0.781113, 1.570796, 1.846274],accel_mss,speed_ms,0,blend_radius_m)
    |   movel([0.275265, -1.315892, -2.614720, -0.781776, 1.570796, 1.846061],accel_mss,speed_ms,0,blend_radius_m)
    |   movel([0.275198, -1.314070, -2.615841, -0.782478, 1.570796, 1.845995],accel_mss,speed_ms,0,blend_radius_m)
    |   movel([0.275231, -1.311845, -2.617203, -0.783340, 1.570796, 1.846028],accel_mss,speed_ms,0,blend_radius_m)
    |   movel([0.275564, -1.307298, -2.619968, -0.785123, 1.570796, 1.846360],accel_mss,speed_ms,0,blend_radius_m)
    |   movel([0.276151, -1.303359, -2.622341, -0.786690, 1.570796, 1.846947],accel_mss,speed_ms,0,blend_radius_m)
    |   movel([0.276989, -1.299497, -2.624648, -0.788245, 1.570796, 1.847786],accel_mss,speed_ms,0,blend_radius_m)
    |   movel([0.278535, -1.293738, -2.628051, -0.790599, 1.570796, 1.849331],accel_mss,speed_ms,0,blend_radius_m)
    |   movel([0.286445, -1.266307, -2.643688, -0.802394, 1.570796, 1.857241],accel_mss,speed_ms,0,blend_radius_m)
    |   movel([0.288606, -1.258326, -2.648062, -0.806001, 1.570796, 1.859402],accel_mss,speed_ms,0,blend_radius_m)
    |   movel([0.289908, -1.252556, -2.651176, -0.808657, 1.570796, 1.860704],accel_mss,speed_ms,0,blend_radius_m)
    |   movel([0.290856, -1.246855, -2.654213, -0.811321, 1.570796, 1.861652],accel_mss,speed_ms,0,blend_radius_m)
    |   movel([0.291357, -1.241212, -2.657182, -0.813996, 1.570796, 1.862153],accel_mss,speed_ms,0,blend_radius_m)
    |   movel([0.291403, -1.238454, -2.658618, -0.815316, 1.570796, 1.862199],accel_mss,speed_ms,0,blend_radius_m)
    |   movel([0.291071, -1.233195, -2.661334, -0.817860, 1.570796, 1.861868],accel_mss,speed_ms,0,blend_radius_m)
    |   movel([0.290684, -1.230708, -2.662607, -0.819074, 1.570796, 1.861481],accel_mss,speed_ms,0,blend_radius_m)
    |   movel([0.289459, -1.225978, -2.665008, -0.821403, 1.570796, 1.860255],accel_mss,speed_ms,0,blend_radius_m)
    |   movel([0.288697, -1.223967, -2.666021, -0.822401, 1.570796, 1.859493],accel_mss,speed_ms,0,blend_radius_m)
    |   movel([0.286729, -1.220259, -2.667877, -0.824253, 1.570796, 1.857525],accel_mss,speed_ms,0,blend_radius_m)
    |   movel([0.285527, -1.218571, -2.668716, -0.825101, 1.570796, 1.856323],accel_mss,speed_ms,0,blend_radius_m)
    |   movel([0.284365, -1.217292, -2.669351, -0.825746, 1.570796, 1.855161],accel_mss,speed_ms,0,blend_radius_m)
    |   movel([0.283014, -1.216195, -2.669893, -0.826301, 1.570796, 1.853810],accel_mss,speed_ms,0,blend_radius_m)
    |   movel([0.281491, -1.215289, -2.670340, -0.826760, 1.570796, 1.852287],accel_mss,speed_ms,0,blend_radius_m)
    |   movel([0.279805, -1.214580, -2.670689, -0.827120, 1.570796, 1.850601],accel_mss,speed_ms,0,blend_radius_m)
    |   movel([0.277838, -1.214135, -2.670908, -0.827346, 1.570796, 1.848635],accel_mss,speed_ms,0,blend_radius_m)
    |   movel([0.275529, -1.214022, -2.670964, -0.827404, 1.570796, 1.846325],accel_mss,speed_ms,0,blend_radius_m)
    |   movel([0.273133, -1.214238, -2.670857, -0.827294, 1.570796, 1.843929],accel_mss,speed_ms,0,blend_radius_m)
    |   movel([0.270926, -1.214776, -2.670593, -0.827021, 1.570796, 1.841723],accel_mss,speed_ms,0,blend_radius_m)
    |   movel([0.269962, -1.215129, -2.670419, -0.826841, 1.570796, 1.840758],accel_mss,speed_ms,0,blend_radius_m)
    |   movel([0.269375, -1.215459, -2.670256, -0.826674, 1.570796, 1.840171],accel_mss,speed_ms,0,blend_radius_m)
    |   movel([0.269070, -1.215798, -2.670089, -0.826502, 1.570796, 1.839867],accel_mss,speed_ms,0,blend_radius_m)
    |   movel([0.268980, -1.216172, -2.669904, -0.826312, 1.570796, 1.839776],accel_mss,speed_ms,0,blend_radius_m)
    |   movel([0.269086, -1.216288, -2.669847, -0.826254, 1.570796, 1.839882],accel_mss,speed_ms,0,blend_radius_m)
    |   movel([0.269364, -1.216293, -2.669845, -0.826251, 1.570796, 1.840160],accel_mss,speed_ms,0,blend_radius_m)
    |   movel([0.270863, -1.215910, -2.670034, -0.826445, 1.570796, 1.841660],accel_mss,speed_ms,0,blend_radius_m)
    |   movel([0.272762, -1.215466, -2.670253, -0.826670, 1.570796, 1.843559],accel_mss,speed_ms,0,blend_radius_m)
    |   movel([0.274581, -1.215256, -2.670356, -0.826777, 1.570796, 1.845378],accel_mss,speed_ms,0,blend_radius_m)
    |   movel([0.276333, -1.215284, -2.670342, -0.826762, 1.570796, 1.847129],accel_mss,speed_ms,0,blend_radius_m)
    |   movel([0.277954, -1.215544, -2.670214, -0.826631, 1.570796, 1.848750],accel_mss,speed_ms,0,blend_radius_m)
    |   movel([0.279558, -1.216058, -2.669961, -0.826370, 1.570796, 1.850355],accel_mss,speed_ms,0,blend_radius_m)
    |   movel([0.280997, -1.216793, -2.669598, -0.825998, 1.570796, 1.851794],accel_mss,speed_ms,0,blend_radius_m)
    |   movel([0.282439, -1.217821, -2.669089, -0.825479, 1.570796, 1.853235],accel_mss,speed_ms,0,blend_radius_m)
    |   movel([0.283729, -1.219007, -2.668500, -0.824882, 1.570796, 1.854525],accel_mss,speed_ms,0,blend_radius_m)
    |   movel([0.285812, -1.221629, -2.667193, -0.823567, 1.570796, 1.856608],accel_mss,speed_ms,0,blend_radius_m)
    |   movel([0.287417, -1.224636, -2.665685, -0.822068, 1.570796, 1.858213],accel_mss,speed_ms,0,blend_radius_m)
    |   movel([0.288694, -1.228258, -2.663854, -0.820277, 1.570796, 1.859491],accel_mss,speed_ms,0,blend_radius_m)
    |   movel([0.289552, -1.232127, -2.661881, -0.818380, 1.570796, 1.860348],accel_mss,speed_ms,0,blend_radius_m)
    |   movel([0.290034, -1.236499, -2.659632, -0.816258, 1.570796, 1.860831],accel_mss,speed_ms,0,blend_radius_m)
    |   movel([0.290100, -1.241048, -2.657267, -0.814074, 1.570796, 1.860896],accel_mss,speed_ms,0,blend_radius_m)
    |   movel([0.289761, -1.245956, -2.654688, -0.811745, 1.570796, 1.860558],accel_mss,speed_ms,0,blend_radius_m)
    |   movel([0.289058, -1.250959, -2.652030, -0.809400, 1.570796, 1.859854],accel_mss,speed_ms,0,blend_radius_m)
    |   movel([0.288525, -1.253670, -2.650578, -0.808142, 1.570796, 1.859321],accel_mss,speed_ms,0,blend_radius_m)
    |   movel([0.286825, -1.260992, -2.646609, -0.804788, 1.570796, 1.857622],accel_mss,speed_ms,0,blend_radius_m)
    |   movel([0.286172, -1.263378, -2.645302, -0.803709, 1.570796, 1.856968],accel_mss,speed_ms,0,blend_radius_m)
    |   movel([0.285602, -1.265093, -2.644358, -0.802938, 1.570796, 1.856398],accel_mss,speed_ms,0,blend_radius_m)
    |   movel([0.285403, -1.265336, -2.644224, -0.802829, 1.570796, 1.856200],accel_mss,speed_ms,0,blend_radius_m)
    |   movel([0.284846, -1.265641, -2.644056, -0.802692, 1.570796, 1.855642],accel_mss,speed_ms,0,blend_radius_m)
    |   movel([0.284553, -1.265918, -2.643902, -0.802568, 1.570796, 1.855349],accel_mss,speed_ms,0,blend_radius_m)
    |   movel([0.283667, -1.267175, -2.643207, -0.802007, 1.570796, 1.854464],accel_mss,speed_ms,0,blend_radius_m)
    |   movel([0.282650, -1.268861, -2.642272, -0.801257, 1.570796, 1.853446],accel_mss,speed_ms,0,blend_radius_m)
    |   movel([0.281743, -1.270594, -2.641306, -0.800489, 1.570796, 1.852539],accel_mss,speed_ms,0,blend_radius_m)
    |   movel([0.280998, -1.272263, -2.640372, -0.799753, 1.570796, 1.851794],accel_mss,speed_ms,0,blend_radius_m)
    |   movel([0.280469, -1.273758, -2.639533, -0.799097, 1.570796, 1.851265],accel_mss,speed_ms,0,blend_radius_m)
    |   movel([0.279985, -1.275386, -2.638617, -0.798386, 1.570796, 1.850781],accel_mss,speed_ms,0,blend_radius_m)
    |   movel([0.279458, -1.275472, -2.638568, -0.798349, 1.570796, 1.850255],accel_mss,speed_ms,0,blend_radius_m)
    |   movel([0.279133, -1.275581, -2.638507, -0.798301, 1.570796, 1.849929],accel_mss,speed_ms,0,blend_radius_m)
    |   movel([0.278874, -1.275781, -2.638394, -0.798214, 1.570796, 1.849670],accel_mss,speed_ms,0,blend_radius_m)
    |   movel([0.278581, -1.276168, -2.638175, -0.798045, 1.570796, 1.849377],accel_mss,speed_ms,0,blend_radius_m)
    |   movel([0.277511, -1.277990, -2.637144, -0.797255, 1.570796, 1.848307],accel_mss,speed_ms,0,blend_radius_m)
    |   movel([0.277141, -1.278782, -2.636694, -0.796913, 1.570796, 1.847937],accel_mss,speed_ms,0,blend_radius_m)
    |   movel([0.276026, -1.282296, -2.634688, -0.795404, 1.570796, 1.846822],accel_mss,speed_ms,0,blend_radius_m)
    |   movel([0.275749, -1.283330, -2.634095, -0.794963, 1.570796, 1.846545],accel_mss,speed_ms,0,blend_radius_m)
    |   movel([0.275335, -1.285324, -2.632948, -0.794116, 1.570796, 1.846132],accel_mss,speed_ms,0,blend_radius_m)
    |   movel([0.274479, -1.284256, -2.633564, -0.794570, 1.570796, 1.845275],accel_mss,speed_ms,0,blend_radius_m)
    |   movel([0.274210, -1.284241, -2.633572, -0.794576, 1.570796, 1.845007],accel_mss,speed_ms,0,blend_radius_m)
    |   movel([0.273843, -1.284416, -2.633471, -0.794501, 1.570796, 1.844639],accel_mss,speed_ms,0,blend_radius_m)
    |   movel([0.273658, -1.284643, -2.633341, -0.794405, 1.570796, 1.844454],accel_mss,speed_ms,0,blend_radius_m)
    |   movel([0.273373, -1.285943, -2.632591, -0.793855, 1.570796, 1.844169],accel_mss,speed_ms,0,blend_radius_m)
    |   movel([0.273169, -1.287545, -2.631664, -0.793179, 1.570796, 1.843966],accel_mss,speed_ms,0,blend_radius_m)
    |   movel([0.272744, -1.292945, -2.628517, -0.790927, 1.570796, 1.843540],accel_mss,speed_ms,0,blend_radius_m)
    |   movel([0.272632, -1.295819, -2.626826, -0.789744, 1.570796, 1.843428],accel_mss,speed_ms,0,blend_radius_m)
    |   movel([0.272636, -1.299145, -2.624857, -0.788387, 1.570796, 1.843432],accel_mss,speed_ms,0,blend_radius_m)
    |   movel([0.271372, -1.297232, -2.625991, -0.789166, 1.570796, 1.842168],accel_mss,speed_ms,0,blend_radius_m)
    |   movel([0.270969, -1.296533, -2.626404, -0.789451, 1.570796, 1.841765],accel_mss,speed_ms,0,blend_radius_m)
    |   movel([0.270589, -1.296185, -2.626610, -0.789594, 1.570796, 1.841385],accel_mss,speed_ms,0,blend_radius_m)
    |   movel([0.270242, -1.296184, -2.626611, -0.789594, 1.570796, 1.841039],accel_mss,speed_ms,0,blend_radius_m)
    |   movel([0.269936, -1.296436, -2.626462, -0.789491, 1.570796, 1.840732],accel_mss,speed_ms,0,blend_radius_m)
    |   movel([0.269778, -1.296832, -2.626228, -0.789329, 1.570796, 1.840575],accel_mss,speed_ms,0,blend_radius_m)
    |   movel([0.269098, -1.301734, -2.623313, -0.787341, 1.570796, 1.839895],accel_mss,speed_ms,0,blend_radius_m)
    |   movel([0.268999, -1.304077, -2.621909, -0.786402, 1.570796, 1.839795],accel_mss,speed_ms,0,blend_radius_m)
    |   movel([0.269093, -1.306514, -2.620442, -0.785433, 1.570796, 1.839889],accel_mss,speed_ms,0,blend_radius_m)
    |   movel([0.269345, -1.308670, -2.619136, -0.784582, 1.570796, 1.840141],accel_mss,speed_ms,0,blend_radius_m)
    |   movel([0.269828, -1.310323, -2.618132, -0.783934, 1.570796, 1.840624],accel_mss,speed_ms,0,blend_radius_m)
    |   movel([0.269880, -1.310531, -2.618005, -0.783853, 1.570796, 1.840676],accel_mss,speed_ms,0,blend_radius_m)
    |   movel([0.269856, -1.310734, -2.617882, -0.783774, 1.570796, 1.840653],accel_mss,speed_ms,0,blend_radius_m)
    |   movel([0.268961, -1.310103, -2.618266, -0.784020, 1.570796, 1.839757],accel_mss,speed_ms,0,blend_radius_m)
    |   movel([0.268104, -1.309533, -2.618612, -0.784243, 1.570796, 1.838900],accel_mss,speed_ms,0,blend_radius_m)
    |   movel([0.267847, -1.309543, -2.618606, -0.784239, 1.570796, 1.838643],accel_mss,speed_ms,0,blend_radius_m)
    |   movel([0.267587, -1.309738, -2.618488, -0.784163, 1.570796, 1.838384],accel_mss,speed_ms,0,blend_radius_m)
    |   movel([0.267387, -1.310096, -2.618270, -0.784023, 1.570796, 1.838183],accel_mss,speed_ms,0,blend_radius_m)
    |   movel([0.267339, -1.310436, -2.618063, -0.783890, 1.570796, 1.838135],accel_mss,speed_ms,0,blend_radius_m)
    |   movel([0.267587, -1.311858, -2.617196, -0.783335, 1.570796, 1.838383],accel_mss,speed_ms,0,blend_radius_m)
    |   movel([0.268092, -1.313474, -2.616207, -0.782708, 1.570796, 1.838889],accel_mss,speed_ms,0,blend_radius_m)
    |   movel([0.268900, -1.315278, -2.615098, -0.782012, 1.570796, 1.839696],accel_mss,speed_ms,0,blend_radius_m)
    |   movel([0.269946, -1.317168, -2.613933, -0.781288, 1.570796, 1.840743],accel_mss,speed_ms,0,blend_radius_m)
    |   movel([0.271186, -1.319050, -2.612768, -0.780571, 1.570796, 1.841983],accel_mss,speed_ms,0,blend_radius_m)
    |   movel([0.271803, -1.319920, -2.612227, -0.780242, 1.570796, 1.842600],accel_mss,speed_ms,0,blend_radius_m)
    |   movel([0.271157, -1.320025, -2.612162, -0.780202, 1.570796, 1.841953],accel_mss,speed_ms,0,blend_radius_m)
    |   movel([0.270474, -1.320067, -2.612136, -0.780186, 1.570796, 1.841271],accel_mss,speed_ms,0,blend_radius_m)
    |   movel([0.269762, -1.319974, -2.612194, -0.780221, 1.570796, 1.840558],accel_mss,speed_ms,0,blend_radius_m)
    |   movel([0.269067, -1.319760, -2.612327, -0.780302, 1.570796, 1.839863],accel_mss,speed_ms,0,blend_radius_m)
    |   movel([0.267809, -1.319118, -2.612726, -0.780546, 1.570796, 1.838605],accel_mss,speed_ms,0,blend_radius_m)
    |   movel([0.267620, -1.319168, -2.612695, -0.780527, 1.570796, 1.838417],accel_mss,speed_ms,0,blend_radius_m)
    |   movel([0.267180, -1.319590, -2.612432, -0.780366, 1.570796, 1.837977],accel_mss,speed_ms,0,blend_radius_m)
    |   movel([0.267124, -1.319845, -2.612274, -0.780270, 1.570796, 1.837921],accel_mss,speed_ms,0,blend_radius_m)
    |   movel([0.267529, -1.321076, -2.611508, -0.779805, 1.570796, 1.838325],accel_mss,speed_ms,0,blend_radius_m)
    |   movel([0.268520, -1.323266, -2.610140, -0.778983, 1.570796, 1.839316],accel_mss,speed_ms,0,blend_radius_m)
    |   movel([0.269611, -1.325030, -2.609033, -0.778325, 1.570796, 1.840408],accel_mss,speed_ms,0,blend_radius_m)
    |   movel([0.270823, -1.326406, -2.608167, -0.777815, 1.570796, 1.841620],accel_mss,speed_ms,0,blend_radius_m)
    |   movel([0.272903, -1.327856, -2.607253, -0.777281, 1.570796, 1.843699],accel_mss,speed_ms,0,blend_radius_m)
    |   movel([0.273069, -1.328019, -2.607149, -0.777221, 1.570796, 1.843865],accel_mss,speed_ms,0,blend_radius_m)
    |   movel([0.273014, -1.328156, -2.607063, -0.777171, 1.570796, 1.843810],accel_mss,speed_ms,0,blend_radius_m)
    |   movel([0.272743, -1.328322, -2.606958, -0.777110, 1.570796, 1.843539],accel_mss,speed_ms,0,blend_radius_m)
    |   movel([0.271501, -1.328673, -2.606735, -0.776981, 1.570796, 1.842297],accel_mss,speed_ms,0,blend_radius_m)
    |   movel([0.270868, -1.328694, -2.606722, -0.776973, 1.570796, 1.841664],accel_mss,speed_ms,0,blend_radius_m)
    |   movel([0.269652, -1.328518, -2.606833, -0.777037, 1.570796, 1.840448],accel_mss,speed_ms,0,blend_radius_m)
    |   movel([0.269466, -1.328590, -2.606788, -0.777011, 1.570796, 1.840262],accel_mss,speed_ms,0,blend_radius_m)
    |   movel([0.269045, -1.328953, -2.606558, -0.776878, 1.570796, 1.839842],accel_mss,speed_ms,0,blend_radius_m)
    |   movel([0.268965, -1.329110, -2.606458, -0.776821, 1.570796, 1.839761],accel_mss,speed_ms,0,blend_radius_m)
    |   movel([0.269090, -1.329618, -2.606136, -0.776635, 1.570796, 1.839886],accel_mss,speed_ms,0,blend_radius_m)
    |   movel([0.269235, -1.329888, -2.605965, -0.776536, 1.570796, 1.840031],accel_mss,speed_ms,0,blend_radius_m)
    |   movel([0.270249, -1.331092, -2.605199, -0.776098, 1.570796, 1.841045],accel_mss,speed_ms,0,blend_radius_m)
    |   movel([0.271477, -1.332013, -2.604612, -0.775763, 1.570796, 1.842273],accel_mss,speed_ms,0,blend_radius_m)
    |   movel([0.273028, -1.332659, -2.604200, -0.775530, 1.570796, 1.843824],accel_mss,speed_ms,0,blend_radius_m)
    |   movel([0.274731, -1.332975, -2.603998, -0.775416, 1.570796, 1.845527],accel_mss,speed_ms,0,blend_radius_m)
    |   movel([0.276743, -1.332874, -2.604063, -0.775452, 1.570796, 1.847539],accel_mss,speed_ms,0,blend_radius_m)
    |   movel([0.277017, -1.332868, -2.604067, -0.775455, 1.570796, 1.847813],accel_mss,speed_ms,0,blend_radius_m)
    |   movel([0.277241, -1.332943, -2.604019, -0.775427, 1.570796, 1.848037],accel_mss,speed_ms,0,blend_radius_m)
    |   movel([0.276956, -1.333267, -2.603812, -0.775311, 1.570796, 1.847752],accel_mss,speed_ms,0,blend_radius_m)
    |   movel([0.275678, -1.333909, -2.603401, -0.775079, 1.570796, 1.846474],accel_mss,speed_ms,0,blend_radius_m)
    |   movel([0.274291, -1.334519, -2.603009, -0.774860, 1.570796, 1.845088],accel_mss,speed_ms,0,blend_radius_m)
    |   movel([0.273098, -1.334926, -2.602749, -0.774715, 1.570796, 1.843895],accel_mss,speed_ms,0,blend_radius_m)
    |   movel([0.271721, -1.335386, -2.602453, -0.774550, 1.570796, 1.842518],accel_mss,speed_ms,0,blend_radius_m)
    |   movel([0.271466, -1.335564, -2.602339, -0.774486, 1.570796, 1.842263],accel_mss,speed_ms,0,blend_radius_m)
    |   movel([0.271327, -1.335814, -2.602178, -0.774397, 1.570796, 1.842123],accel_mss,speed_ms,0,blend_radius_m)
    |   movel([0.271343, -1.336074, -2.602011, -0.774304, 1.570796, 1.842139],accel_mss,speed_ms,0,blend_radius_m)
    |   movel([0.271507, -1.336238, -2.601905, -0.774245, 1.570796, 1.842303],accel_mss,speed_ms,0,blend_radius_m)
    |   movel([0.272716, -1.336703, -2.601606, -0.774080, 1.570796, 1.843512],accel_mss,speed_ms,0,blend_radius_m)
    |   movel([0.274047, -1.337050, -2.601382, -0.773957, 1.570796, 1.844843],accel_mss,speed_ms,0,blend_radius_m)
    |   movel([0.275300, -1.337202, -2.601284, -0.773902, 1.570796, 1.846096],accel_mss,speed_ms,0,blend_radius_m)
    |   movel([0.276678, -1.337172, -2.601304, -0.773913, 1.570796, 1.847474],accel_mss,speed_ms,0,blend_radius_m)
    |   movel([0.278384, -1.336966, -2.601437, -0.773987, 1.570796, 1.849180],accel_mss,speed_ms,0,blend_radius_m)
    |   movel([0.279266, -1.336820, -2.601530, -0.774038, 1.570796, 1.850062],accel_mss,speed_ms,0,blend_radius_m)
    |   movel([0.281169, -1.336390, -2.601807, -0.774191, 1.570796, 1.851966],accel_mss,speed_ms,0,blend_radius_m)
    |   movel([0.281589, -1.336173, -2.601948, -0.774269, 1.570796, 1.852385],accel_mss,speed_ms,0,blend_radius_m)
    |   movel([0.281862, -1.335916, -2.602113, -0.774361, 1.570796, 1.852658],accel_mss,speed_ms,0,blend_radius_m)
    |   movel([0.281947, -1.335663, -2.602275, -0.774451, 1.570796, 1.852743],accel_mss,speed_ms,0,blend_radius_m)
    |   movel([0.281691, -1.335396, -2.602447, -0.774546, 1.570796, 1.852488],accel_mss,speed_ms,0,blend_radius_m)
    |   movel([0.281436, -1.335403, -2.602442, -0.774543, 1.570796, 1.852232],accel_mss,speed_ms,0,blend_radius_m)
    |   movel([0.280605, -1.335608, -2.602311, -0.774471, 1.570796, 1.851402],accel_mss,speed_ms,0,blend_radius_m)
    |   speed_ms = 0.005
    |   movel([0.280605, -1.326609, -2.598112, -0.787668, 1.570796, 1.851402],accel_mss,speed_ms,0,blend_radius_m)
    |   speed_ms = 0.040
    |   # Splitting Linear movement in 2 (instruction 6735: MoveL 6486)
    |   movel([0.250414, -1.344809, -2.586346, -0.781234, 1.570796, 1.821210],accel_mss,speed_ms,0,blend_radius_m)
    |   movel([0.221110, -1.362951, -2.574168, -0.775271, 1.570796, 1.791906],accel_mss,speed_ms,0,blend_radius_m)
    |   speed_ms = 0.005
    |   movel([0.221110, -1.371710, -2.578207, -0.762473, 1.570796, 1.791906],accel_mss,speed_ms,0,blend_radius_m)
    |   speed_ms = 0.025
    |   movel([0.221643, -1.370422, -2.579098, -0.762869, 1.570796, 1.792439],accel_mss,speed_ms,0,blend_radius_m)
    |   movel([0.222388, -1.367982, -2.580780, -0.763627, 1.570796, 1.793184],accel_mss,speed_ms,0,blend_radius_m)
    |   movel([0.222534, -1.367034, -2.581431, -0.763923, 1.570796, 1.793331],accel_mss,speed_ms,0,blend_radius_m)
    |   movel([0.222561, -1.365826, -2.582260, -0.764304, 1.570796, 1.793358],accel_mss,speed_ms,0,blend_radius_m)
    |   movel([0.222436, -1.364673, -2.583048, -0.764668, 1.570796, 1.793232],accel_mss,speed_ms,0,blend_radius_m)
    |   movel([0.222163, -1.363610, -2.583773, -0.765006, 1.570796, 1.792959],accel_mss,speed_ms,0,blend_radius_m)
    |   movel([0.221737, -1.362632, -2.584439, -0.765318, 1.570796, 1.792533],accel_mss,speed_ms,0,blend_radius_m)
    |   movel([0.221193, -1.361803, -2.585002, -0.765584, 1.570796, 1.791990],accel_mss,speed_ms,0,blend_radius_m)
    |   movel([0.220511, -1.361087, -2.585488, -0.765814, 1.570796, 1.791307],accel_mss,speed_ms,0,blend_radius_m)
    |   movel([0.219749, -1.360562, -2.585844, -0.765983, 1.570796, 1.790545],accel_mss,speed_ms,0,blend_radius_m)
    |   movel([0.218849, -1.360194, -2.586093, -0.766102, 1.570796, 1.789646],accel_mss,speed_ms,0,blend_radius_m)
    |   movel([0.217588, -1.359980, -2.586238, -0.766171, 1.570796, 1.788384],accel_mss,speed_ms,0,blend_radius_m)
    |   movel([0.216186, -1.360043, -2.586195, -0.766151, 1.570796, 1.786983],accel_mss,speed_ms,0,blend_radius_m)
    |   movel([0.214719, -1.360378, -2.585968, -0.766042, 1.570796, 1.785516],accel_mss,speed_ms,0,blend_radius_m)
    |   movel([0.213233, -1.360981, -2.585560, -0.765848, 1.570796, 1.784030],accel_mss,speed_ms,0,blend_radius_m)
    |   movel([0.211826, -1.361803, -2.585002, -0.765584, 1.570796, 1.782623],accel_mss,speed_ms,0,blend_radius_m)
    |   movel([0.210530, -1.362827, -2.584306, -0.765256, 1.570796, 1.781326],accel_mss,speed_ms,0,blend_radius_m)
    |   movel([0.209427, -1.363988, -2.583515, -0.764886, 1.570796, 1.780223],accel_mss,speed_ms,0,blend_radius_m)
    |   movel([0.208554, -1.365246, -2.582656, -0.764487, 1.570796, 1.779350],accel_mss,speed_ms,0,blend_radius_m)
    |   movel([0.208218, -1.365899, -2.582209, -0.764280, 1.570796, 1.779014],accel_mss,speed_ms,0,blend_radius_m)
    |   movel([0.208036, -1.366437, -2.581841, -0.764111, 1.570796, 1.778832],accel_mss,speed_ms,0,blend_radius_m)
    |   movel([0.208014, -1.366809, -2.581586, -0.763994, 1.570796, 1.778810],accel_mss,speed_ms,0,blend_radius_m)
    |   movel([0.208165, -1.366960, -2.581482, -0.763947, 1.570796, 1.778962],accel_mss,speed_ms,0,blend_radius_m)
    |   movel([0.208440, -1.366917, -2.581512, -0.763960, 1.570796, 1.779237],accel_mss,speed_ms,0,blend_radius_m)
    |   movel([0.208737, -1.366729, -2.581641, -0.764019, 1.570796, 1.779534],accel_mss,speed_ms,0,blend_radius_m)
    |   movel([0.208988, -1.366432, -2.581844, -0.764113, 1.570796, 1.779784],accel_mss,speed_ms,0,blend_radius_m)
    |   movel([0.209129, -1.366105, -2.582068, -0.764216, 1.570796, 1.779925],accel_mss,speed_ms,0,blend_radius_m)
    |   movel([0.209548, -1.365201, -2.582687, -0.764501, 1.570796, 1.780344],accel_mss,speed_ms,0,blend_radius_m)
    |   movel([0.210459, -1.364080, -2.583453, -0.764856, 1.570796, 1.781255],accel_mss,speed_ms,0,blend_radius_m)
    |   movel([0.211639, -1.362966, -2.584211, -0.765211, 1.570796, 1.782435],accel_mss,speed_ms,0,blend_radius_m)
    |   movel([0.212893, -1.362072, -2.584820, -0.765497, 1.570796, 1.783689],accel_mss,speed_ms,0,blend_radius_m)
    |   movel([0.213501, -1.361734, -2.585049, -0.765606, 1.570796, 1.784298],accel_mss,speed_ms,0,blend_radius_m)
    |   movel([0.214009, -1.361515, -2.585198, -0.765676, 1.570796, 1.784805],accel_mss,speed_ms,0,blend_radius_m)
    |   movel([0.216451, -1.360992, -2.585553, -0.765845, 1.570796, 1.787247],accel_mss,speed_ms,0,blend_radius_m)
    |   movel([0.217029, -1.360941, -2.585587, -0.765861, 1.570796, 1.787826],accel_mss,speed_ms,0,blend_radius_m)
    |   movel([0.218102, -1.361120, -2.585466, -0.765803, 1.570796, 1.788898],accel_mss,speed_ms,0,blend_radius_m)
    |   movel([0.218824, -1.361405, -2.585272, -0.765711, 1.570796, 1.789620],accel_mss,speed_ms,0,blend_radius_m)
    |   movel([0.219441, -1.361814, -2.584995, -0.765580, 1.570796, 1.790238],accel_mss,speed_ms,0,blend_radius_m)
    |   movel([0.220023, -1.362385, -2.584607, -0.765397, 1.570796, 1.790820],accel_mss,speed_ms,0,blend_radius_m)
    |   movel([0.220904, -1.363803, -2.583642, -0.764944, 1.570796, 1.791700],accel_mss,speed_ms,0,blend_radius_m)
    |   movel([0.221191, -1.364638, -2.583072, -0.764679, 1.570796, 1.791987],accel_mss,speed_ms,0,blend_radius_m)
    |   movel([0.221418, -1.366460, -2.581825, -0.764104, 1.570796, 1.792214],accel_mss,speed_ms,0,blend_radius_m)
    |   movel([0.221275, -1.367961, -2.580795, -0.763634, 1.570796, 1.792071],accel_mss,speed_ms,0,blend_radius_m)
    |   movel([0.220853, -1.369678, -2.579612, -0.763099, 1.570796, 1.791649],accel_mss,speed_ms,0,blend_radius_m)
    |   movel([0.220207, -1.371436, -2.578396, -0.762557, 1.570796, 1.791004],accel_mss,speed_ms,0,blend_radius_m)
    |   movel([0.219395, -1.373060, -2.577269, -0.762059, 1.570796, 1.790191],accel_mss,speed_ms,0,blend_radius_m)
    |   movel([0.217960, -1.375339, -2.575682, -0.761368, 1.570796, 1.788756],accel_mss,speed_ms,0,blend_radius_m)
    |   movel([0.216413, -1.377377, -2.574256, -0.760755, 1.570796, 1.787209],accel_mss,speed_ms,0,blend_radius_m)
    |   movel([0.214666, -1.379290, -2.572913, -0.760186, 1.570796, 1.785463],accel_mss,speed_ms,0,blend_radius_m)
    |   movel([0.211114, -1.382550, -2.570611, -0.759228, 1.570796, 1.781911],accel_mss,speed_ms,0,blend_radius_m)
    |   movel([0.210870, -1.382858, -2.570392, -0.759139, 1.570796, 1.781666],accel_mss,speed_ms,0,blend_radius_m)
    |   movel([0.210841, -1.383051, -2.570256, -0.759083, 1.570796, 1.781637],accel_mss,speed_ms,0,blend_radius_m)
    |   movel([0.211032, -1.383224, -2.570133, -0.759032, 1.570796, 1.781829],accel_mss,speed_ms,0,blend_radius_m)
    |   movel([0.211291, -1.383202, -2.570149, -0.759039, 1.570796, 1.782087],accel_mss,speed_ms,0,blend_radius_m)
    |   movel([0.211723, -1.382941, -2.570333, -0.759114, 1.570796, 1.782519],accel_mss,speed_ms,0,blend_radius_m)
    |   movel([0.213964, -1.381122, -2.571621, -0.759646, 1.570796, 1.784760],accel_mss,speed_ms,0,blend_radius_m)
    |   movel([0.215188, -1.379957, -2.572443, -0.759989, 1.570796, 1.785985],accel_mss,speed_ms,0,blend_radius_m)
    |   movel([0.216423, -1.378644, -2.573367, -0.760378, 1.570796, 1.787219],accel_mss,speed_ms,0,blend_radius_m)
    |   movel([0.217577, -1.377284, -2.574322, -0.760783, 1.570796, 1.788373],accel_mss,speed_ms,0,blend_radius_m)
    |   movel([0.219620, -1.374450, -2.576303, -0.761637, 1.570796, 1.790417],accel_mss,speed_ms,0,blend_radius_m)
    |   movel([0.220428, -1.373087, -2.577251, -0.762051, 1.570796, 1.791224],accel_mss,speed_ms,0,blend_radius_m)
    |   movel([0.221110, -1.371710, -2.578207, -0.762473, 1.570796, 1.791906],accel_mss,speed_ms,0,blend_radius_m)
    |   movel([0.221643, -1.370422, -2.579098, -0.762869, 1.570796, 1.792439],accel_mss,speed_ms,0,blend_radius_m)
    |   movel([0.221952, -1.369409, -2.579797, -0.763183, 1.570796, 1.792749],accel_mss,speed_ms,0,blend_radius_m)
    |   speed_ms = 0.005
    |   movel([0.221952, -1.360634, -2.575748, -0.776007, 1.570796, 1.792749],accel_mss,speed_ms,0,blend_radius_m)
    |   speed_ms = 0.040
    |   # Splitting Linear movement in 2 (instruction 6806: MoveL 6553)
    |   movel([0.232507, -1.336732, -2.591623, -0.784034, 1.570796, 1.803303],accel_mss,speed_ms,0,blend_radius_m)
    |   movel([0.243637, -1.311871, -2.607315, -0.793203, 1.570796, 1.814433],accel_mss,speed_ms,0,blend_radius_m)
    |   speed_ms = 0.005
    |   movel([0.243637, -1.320960, -2.611580, -0.779849, 1.570796, 1.814433],accel_mss,speed_ms,0,blend_radius_m)
    |   speed_ms = 0.025
    |   movel([0.241436, -1.324397, -2.609431, -0.778561, 1.570796, 1.812232],accel_mss,speed_ms,0,blend_radius_m)
    |   movel([0.239068, -1.327689, -2.607358, -0.777342, 1.570796, 1.809864],accel_mss,speed_ms,0,blend_radius_m)
    |   movel([0.236650, -1.330694, -2.605453, -0.776243, 1.570796, 1.807447],accel_mss,speed_ms,0,blend_radius_m)
    |   movel([0.234288, -1.333264, -2.603814, -0.775312, 1.570796, 1.805085],accel_mss,speed_ms,0,blend_radius_m)
    |   movel([0.232683, -1.334753, -2.602860, -0.774776, 1.570796, 1.803480],accel_mss,speed_ms,0,blend_radius_m)
    |   movel([0.232322, -1.334895, -2.602769, -0.774726, 1.570796, 1.803119],accel_mss,speed_ms,0,blend_radius_m)
    |   movel([0.232040, -1.334813, -2.602821, -0.774755, 1.570796, 1.802837],accel_mss,speed_ms,0,blend_radius_m)
    |   movel([0.231965, -1.334654, -2.602923, -0.774812, 1.570796, 1.802762],accel_mss,speed_ms,0,blend_radius_m)
    |   movel([0.232167, -1.334130, -2.603259, -0.775000, 1.570796, 1.802964],accel_mss,speed_ms,0,blend_radius_m)
    |   movel([0.232601, -1.333473, -2.603680, -0.775236, 1.570796, 1.803397],accel_mss,speed_ms,0,blend_radius_m)
    |   movel([0.233282, -1.332300, -2.604429, -0.775660, 1.570796, 1.804079],accel_mss,speed_ms,0,blend_radius_m)
    |   movel([0.233567, -1.331678, -2.604826, -0.775885, 1.570796, 1.804363],accel_mss,speed_ms,0,blend_radius_m)
    |   movel([0.234233, -1.329789, -2.606028, -0.776572, 1.570796, 1.805030],accel_mss,speed_ms,0,blend_radius_m)
    |   movel([0.232756, -1.331325, -2.605051, -0.776013, 1.570796, 1.803552],accel_mss,speed_ms,0,blend_radius_m)
    |   movel([0.230117, -1.333800, -2.603470, -0.775118, 1.570796, 1.800913],accel_mss,speed_ms,0,blend_radius_m)
    |   movel([0.227069, -1.336172, -2.601948, -0.774269, 1.570796, 1.797866],accel_mss,speed_ms,0,blend_radius_m)
    |   movel([0.223823, -1.338288, -2.600583, -0.773518, 1.570796, 1.794620],accel_mss,speed_ms,0,blend_radius_m)
    |   movel([0.222214, -1.339193, -2.599998, -0.773198, 1.570796, 1.793010],accel_mss,speed_ms,0,blend_radius_m)
    |   movel([0.219498, -1.340494, -2.599154, -0.772741, 1.570796, 1.790294],accel_mss,speed_ms,0,blend_radius_m)
    |   movel([0.218879, -1.340680, -2.599033, -0.772676, 1.570796, 1.789675],accel_mss,speed_ms,0,blend_radius_m)
    |   movel([0.218585, -1.340627, -2.599068, -0.772694, 1.570796, 1.789381],accel_mss,speed_ms,0,blend_radius_m)
    |   movel([0.218517, -1.340378, -2.599229, -0.772782, 1.570796, 1.789313],accel_mss,speed_ms,0,blend_radius_m)
    |   movel([0.218961, -1.339700, -2.599669, -0.773020, 1.570796, 1.789757],accel_mss,speed_ms,0,blend_radius_m)
    |   movel([0.219188, -1.339478, -2.599813, -0.773098, 1.570796, 1.789985],accel_mss,speed_ms,0,blend_radius_m)
    |   movel([0.219992, -1.338747, -2.600286, -0.773356, 1.570796, 1.790788],accel_mss,speed_ms,0,blend_radius_m)
    |   movel([0.219999, -1.338594, -2.600386, -0.773410, 1.570796, 1.790796],accel_mss,speed_ms,0,blend_radius_m)
    |   movel([0.219711, -1.338646, -2.600352, -0.773391, 1.570796, 1.790508],accel_mss,speed_ms,0,blend_radius_m)
    |   movel([0.218535, -1.339304, -2.599926, -0.773159, 1.570796, 1.789332],accel_mss,speed_ms,0,blend_radius_m)
    |   movel([0.215771, -1.340688, -2.599028, -0.772673, 1.570796, 1.786567],accel_mss,speed_ms,0,blend_radius_m)
    |   movel([0.212874, -1.341760, -2.598331, -0.772298, 1.570796, 1.783670],accel_mss,speed_ms,0,blend_radius_m)
    |   movel([0.210546, -1.342336, -2.597955, -0.772097, 1.570796, 1.781343],accel_mss,speed_ms,0,blend_radius_m)
    |   movel([0.210170, -1.342256, -2.598008, -0.772125, 1.570796, 1.780967],accel_mss,speed_ms,0,blend_radius_m)
    |   movel([0.210090, -1.341905, -2.598236, -0.772248, 1.570796, 1.780886],accel_mss,speed_ms,0,blend_radius_m)
    |   movel([0.210162, -1.341776, -2.598321, -0.772293, 1.570796, 1.780958],accel_mss,speed_ms,0,blend_radius_m)
    |   movel([0.211755, -1.340343, -2.599252, -0.772794, 1.570796, 1.782552],accel_mss,speed_ms,0,blend_radius_m)
    |   movel([0.212058, -1.340015, -2.599465, -0.772909, 1.570796, 1.782855],accel_mss,speed_ms,0,blend_radius_m)
    |   movel([0.212074, -1.339865, -2.599562, -0.772962, 1.570796, 1.782870],accel_mss,speed_ms,0,blend_radius_m)
    |   movel([0.211898, -1.339829, -2.599586, -0.772975, 1.570796, 1.782694],accel_mss,speed_ms,0,blend_radius_m)
    |   movel([0.211329, -1.339855, -2.599569, -0.772965, 1.570796, 1.782125],accel_mss,speed_ms,0,blend_radius_m)
    |   movel([0.210090, -1.339663, -2.599693, -0.773033, 1.570796, 1.780886],accel_mss,speed_ms,0,blend_radius_m)
    |   movel([0.208885, -1.339424, -2.599848, -0.773117, 1.570796, 1.779681],accel_mss,speed_ms,0,blend_radius_m)
    |   movel([0.208347, -1.339206, -2.599989, -0.773194, 1.570796, 1.779143],accel_mss,speed_ms,0,blend_radius_m)
    |   movel([0.208024, -1.338909, -2.600181, -0.773298, 1.570796, 1.778820],accel_mss,speed_ms,0,blend_radius_m)
    |   movel([0.208057, -1.338776, -2.600268, -0.773345, 1.570796, 1.778853],accel_mss,speed_ms,0,blend_radius_m)
    |   movel([0.208644, -1.338217, -2.600629, -0.773543, 1.570796, 1.779440],accel_mss,speed_ms,0,blend_radius_m)
    |   movel([0.208934, -1.338007, -2.600765, -0.773617, 1.570796, 1.779730],accel_mss,speed_ms,0,blend_radius_m)
    |   movel([0.209893, -1.337408, -2.601151, -0.773829, 1.570796, 1.780690],accel_mss,speed_ms,0,blend_radius_m)
    |   movel([0.209020, -1.337141, -2.601324, -0.773924, 1.570796, 1.779816],accel_mss,speed_ms,0,blend_radius_m)
    |   movel([0.207611, -1.336506, -2.601733, -0.774150, 1.570796, 1.778407],accel_mss,speed_ms,0,blend_radius_m)
    |   movel([0.207285, -1.336171, -2.601948, -0.774269, 1.570796, 1.778081],accel_mss,speed_ms,0,blend_radius_m)
    |   movel([0.207309, -1.335873, -2.602140, -0.774376, 1.570796, 1.778105],accel_mss,speed_ms,0,blend_radius_m)
    |   movel([0.207563, -1.335618, -2.602304, -0.774467, 1.570796, 1.778359],accel_mss,speed_ms,0,blend_radius_m)
    |   movel([0.207887, -1.335508, -2.602375, -0.774506, 1.570796, 1.778683],accel_mss,speed_ms,0,blend_radius_m)
    |   movel([0.208323, -1.335566, -2.602337, -0.774485, 1.570796, 1.779120],accel_mss,speed_ms,0,blend_radius_m)
    |   movel([0.209653, -1.336069, -2.602014, -0.774306, 1.570796, 1.780449],accel_mss,speed_ms,0,blend_radius_m)
    |   movel([0.210624, -1.336278, -2.601880, -0.774231, 1.570796, 1.781421],accel_mss,speed_ms,0,blend_radius_m)
    |   movel([0.211587, -1.336408, -2.601796, -0.774185, 1.570796, 1.782383],accel_mss,speed_ms,0,blend_radius_m)
    |   movel([0.212178, -1.336370, -2.601821, -0.774199, 1.570796, 1.782974],accel_mss,speed_ms,0,blend_radius_m)
    |   movel([0.212366, -1.336431, -2.601781, -0.774177, 1.570796, 1.783162],accel_mss,speed_ms,0,blend_radius_m)
    |   movel([0.212370, -1.336562, -2.601697, -0.774130, 1.570796, 1.783166],accel_mss,speed_ms,0,blend_radius_m)
    |   movel([0.212167, -1.337049, -2.601383, -0.773957, 1.570796, 1.782963],accel_mss,speed_ms,0,blend_radius_m)
    |   movel([0.211962, -1.337261, -2.601246, -0.773882, 1.570796, 1.782758],accel_mss,speed_ms,0,blend_radius_m)
    |   movel([0.210250, -1.338157, -2.600668, -0.773564, 1.570796, 1.781046],accel_mss,speed_ms,0,blend_radius_m)
    |   movel([0.210020, -1.338306, -2.600571, -0.773511, 1.570796, 1.780817],accel_mss,speed_ms,0,blend_radius_m)
    |   movel([0.210096, -1.338533, -2.600425, -0.773431, 1.570796, 1.780892],accel_mss,speed_ms,0,blend_radius_m)
    |   movel([0.211313, -1.338743, -2.600289, -0.773357, 1.570796, 1.782109],accel_mss,speed_ms,0,blend_radius_m)
    |   movel([0.212322, -1.338808, -2.600247, -0.773334, 1.570796, 1.783118],accel_mss,speed_ms,0,blend_radius_m)
    |   movel([0.213867, -1.338890, -2.600194, -0.773305, 1.570796, 1.784664],accel_mss,speed_ms,0,blend_radius_m)
    |   movel([0.214020, -1.339106, -2.600054, -0.773229, 1.570796, 1.784817],accel_mss,speed_ms,0,blend_radius_m)
    |   movel([0.213861, -1.339480, -2.599812, -0.773097, 1.570796, 1.784657],accel_mss,speed_ms,0,blend_radius_m)
    |   movel([0.213314, -1.340089, -2.599417, -0.772883, 1.570796, 1.784111],accel_mss,speed_ms,0,blend_radius_m)
    |   movel([0.212588, -1.340817, -2.598944, -0.772628, 1.570796, 1.783384],accel_mss,speed_ms,0,blend_radius_m)
    |   movel([0.213222, -1.340688, -2.599028, -0.772673, 1.570796, 1.784019],accel_mss,speed_ms,0,blend_radius_m)
    |   movel([0.214875, -1.340168, -2.599366, -0.772856, 1.570796, 1.785672],accel_mss,speed_ms,0,blend_radius_m)
    |   movel([0.217057, -1.339138, -2.600033, -0.773218, 1.570796, 1.787853],accel_mss,speed_ms,0,blend_radius_m)
    |   movel([0.219334, -1.337839, -2.600873, -0.773677, 1.570796, 1.790130],accel_mss,speed_ms,0,blend_radius_m)
    |   movel([0.221318, -1.336464, -2.601760, -0.774165, 1.570796, 1.792115],accel_mss,speed_ms,0,blend_radius_m)
    |   movel([0.222834, -1.335413, -2.602436, -0.774540, 1.570796, 1.793631],accel_mss,speed_ms,0,blend_radius_m)
    |   movel([0.223127, -1.335366, -2.602466, -0.774557, 1.570796, 1.793923],accel_mss,speed_ms,0,blend_radius_m)
    |   movel([0.223280, -1.335523, -2.602365, -0.774501, 1.570796, 1.794077],accel_mss,speed_ms,0,blend_radius_m)
    |   movel([0.223204, -1.335832, -2.602167, -0.774390, 1.570796, 1.794001],accel_mss,speed_ms,0,blend_radius_m)
    |   movel([0.222081, -1.337496, -2.601095, -0.773798, 1.570796, 1.792877],accel_mss,speed_ms,0,blend_radius_m)
    |   movel([0.221431, -1.338294, -2.600579, -0.773515, 1.570796, 1.792227],accel_mss,speed_ms,0,blend_radius_m)
    |   movel([0.220938, -1.338857, -2.600215, -0.773317, 1.570796, 1.791734],accel_mss,speed_ms,0,blend_radius_m)
    |   movel([0.221411, -1.338650, -2.600349, -0.773390, 1.570796, 1.792207],accel_mss,speed_ms,0,blend_radius_m)
    |   movel([0.222438, -1.338128, -2.600687, -0.773574, 1.570796, 1.793234],accel_mss,speed_ms,0,blend_radius_m)
    |   movel([0.224025, -1.337178, -2.601300, -0.773911, 1.570796, 1.794822],accel_mss,speed_ms,0,blend_radius_m)
    |   movel([0.227102, -1.335132, -2.602616, -0.774641, 1.570796, 1.797898],accel_mss,speed_ms,0,blend_radius_m)
    |   movel([0.228730, -1.333855, -2.603436, -0.775099, 1.570796, 1.799526],accel_mss,speed_ms,0,blend_radius_m)
    |   movel([0.230524, -1.332285, -2.604439, -0.775665, 1.570796, 1.801320],accel_mss,speed_ms,0,blend_radius_m)
    |   movel([0.232241, -1.330648, -2.605482, -0.776259, 1.570796, 1.803037],accel_mss,speed_ms,0,blend_radius_m)
    |   movel([0.234795, -1.327983, -2.607172, -0.777234, 1.570796, 1.805591],accel_mss,speed_ms,0,blend_radius_m)
    |   movel([0.235103, -1.327816, -2.607278, -0.777296, 1.570796, 1.805900],accel_mss,speed_ms,0,blend_radius_m)
    |   movel([0.235369, -1.327851, -2.607256, -0.777283, 1.570796, 1.806166],accel_mss,speed_ms,0,blend_radius_m)
    |   movel([0.235545, -1.328095, -2.607101, -0.777193, 1.570796, 1.806341],accel_mss,speed_ms,0,blend_radius_m)
    |   movel([0.235550, -1.328438, -2.606884, -0.777067, 1.570796, 1.806347],accel_mss,speed_ms,0,blend_radius_m)
    |   movel([0.235096, -1.330215, -2.605757, -0.776417, 1.570796, 1.805892],accel_mss,speed_ms,0,blend_radius_m)
    |   movel([0.234806, -1.331255, -2.605096, -0.776038, 1.570796, 1.805603],accel_mss,speed_ms,0,blend_radius_m)
    |   movel([0.234934, -1.331334, -2.605045, -0.776010, 1.570796, 1.805730],accel_mss,speed_ms,0,blend_radius_m)
    |   movel([0.235238, -1.331111, -2.605187, -0.776091, 1.570796, 1.806035],accel_mss,speed_ms,0,blend_radius_m)
    |   movel([0.236484, -1.329635, -2.606126, -0.776629, 1.570796, 1.807280],accel_mss,speed_ms,0,blend_radius_m)
    |   movel([0.238218, -1.327441, -2.607514, -0.777433, 1.570796, 1.809015],accel_mss,speed_ms,0,blend_radius_m)
    |   movel([0.240066, -1.324858, -2.609141, -0.778389, 1.570796, 1.810862],accel_mss,speed_ms,0,blend_radius_m)
    |   movel([0.241891, -1.322091, -2.610875, -0.779423, 1.570796, 1.812687],accel_mss,speed_ms,0,blend_radius_m)
    |   movel([0.243555, -1.319336, -2.612590, -0.780463, 1.570796, 1.814352],accel_mss,speed_ms,0,blend_radius_m)
    |   movel([0.244161, -1.318330, -2.613214, -0.780845, 1.570796, 1.814958],accel_mss,speed_ms,0,blend_radius_m)
    |   movel([0.244571, -1.317812, -2.613535, -0.781042, 1.570796, 1.815368],accel_mss,speed_ms,0,blend_radius_m)
    |   movel([0.244929, -1.317578, -2.613680, -0.781131, 1.570796, 1.815725],accel_mss,speed_ms,0,blend_radius_m)
    |   movel([0.245306, -1.317533, -2.613707, -0.781148, 1.570796, 1.816102],accel_mss,speed_ms,0,blend_radius_m)
    |   movel([0.245425, -1.317704, -2.613602, -0.781083, 1.570796, 1.816221],accel_mss,speed_ms,0,blend_radius_m)
    |   movel([0.245309, -1.318092, -2.613361, -0.780935, 1.570796, 1.816106],accel_mss,speed_ms,0,blend_radius_m)
    |   movel([0.243637, -1.320960, -2.611580, -0.779849, 1.570796, 1.814433],accel_mss,speed_ms,0,blend_radius_m)
    |   movel([0.242061, -1.323421, -2.610043, -0.778925, 1.570796, 1.812857],accel_mss,speed_ms,0,blend_radius_m)
    |   speed_ms = 0.005
    |   movel([0.242061, -1.314347, -2.605789, -0.792253, 1.570796, 1.812857],accel_mss,speed_ms,0,blend_radius_m)
    |   speed_ms = 0.040
    |   movel([0.249676, -1.297935, -2.615756, -0.798698, 1.570796, 1.820473],accel_mss,speed_ms,0,blend_radius_m)
    |   speed_ms = 0.005
    |   movel([0.249676, -1.307108, -2.620083, -0.785198, 1.570796, 1.820473],accel_mss,speed_ms,0,blend_radius_m)
    |   speed_ms = 0.025
    |   movel([0.248671, -1.309163, -2.618837, -0.784389, 1.570796, 1.819468],accel_mss,speed_ms,0,blend_radius_m)
    |   movel([0.247477, -1.311194, -2.617601, -0.783594, 1.570796, 1.818273],accel_mss,speed_ms,0,blend_radius_m)
    |   movel([0.246033, -1.313315, -2.616304, -0.782770, 1.570796, 1.816829],accel_mss,speed_ms,0,blend_radius_m)
    |   movel([0.244447, -1.315381, -2.615035, -0.781973, 1.570796, 1.815244],accel_mss,speed_ms,0,blend_radius_m)
    |   movel([0.242606, -1.317535, -2.613706, -0.781148, 1.570796, 1.813402],accel_mss,speed_ms,0,blend_radius_m)
    |   movel([0.240647, -1.319608, -2.612421, -0.780360, 1.570796, 1.811443],accel_mss,speed_ms,0,blend_radius_m)
    |   movel([0.238434, -1.321752, -2.611086, -0.779550, 1.570796, 1.809230],accel_mss,speed_ms,0,blend_radius_m)
    |   movel([0.236139, -1.323808, -2.609800, -0.778780, 1.570796, 1.806935],accel_mss,speed_ms,0,blend_radius_m)
    |   movel([0.229914, -1.329053, -2.606495, -0.776842, 1.570796, 1.800711],accel_mss,speed_ms,0,blend_radius_m)
    |   movel([0.227745, -1.330774, -2.605402, -0.776213, 1.570796, 1.798541],accel_mss,speed_ms,0,blend_radius_m)
    |   movel([0.225526, -1.332407, -2.604361, -0.775621, 1.570796, 1.796323],accel_mss,speed_ms,0,blend_radius_m)
    |   movel([0.223819, -1.333549, -2.603631, -0.775209, 1.570796, 1.794616],accel_mss,speed_ms,0,blend_radius_m)
    |   movel([0.222076, -1.334582, -2.602969, -0.774838, 1.570796, 1.792872],accel_mss,speed_ms,0,blend_radius_m)
    |   movel([0.220539, -1.335351, -2.602476, -0.774562, 1.570796, 1.791336],accel_mss,speed_ms,0,blend_radius_m)
    |   movel([0.218987, -1.335957, -2.602086, -0.774346, 1.570796, 1.789784],accel_mss,speed_ms,0,blend_radius_m)
    |   movel([0.217718, -1.336295, -2.601869, -0.774225, 1.570796, 1.788514],accel_mss,speed_ms,0,blend_radius_m)
    |   movel([0.216497, -1.336441, -2.601775, -0.774173, 1.570796, 1.787294],accel_mss,speed_ms,0,blend_radius_m)
    |   movel([0.215411, -1.336384, -2.601811, -0.774193, 1.570796, 1.786207],accel_mss,speed_ms,0,blend_radius_m)
    |   movel([0.214451, -1.336114, -2.601985, -0.774290, 1.570796, 1.785248],accel_mss,speed_ms,0,blend_radius_m)
    |   movel([0.213533, -1.335602, -2.602314, -0.774473, 1.570796, 1.784329],accel_mss,speed_ms,0,blend_radius_m)
    |   movel([0.212789, -1.334911, -2.602758, -0.774720, 1.570796, 1.783585],accel_mss,speed_ms,0,blend_radius_m)
    |   movel([0.212047, -1.333896, -2.603409, -0.775084, 1.570796, 1.782843],accel_mss,speed_ms,0,blend_radius_m)
    |   movel([0.210223, -1.330600, -2.605512, -0.776277, 1.570796, 1.781019],accel_mss,speed_ms,0,blend_radius_m)
    |   movel([0.209733, -1.329987, -2.605902, -0.776500, 1.570796, 1.780530],accel_mss,speed_ms,0,blend_radius_m)
    |   movel([0.209476, -1.330037, -2.605870, -0.776482, 1.570796, 1.780272],accel_mss,speed_ms,0,blend_radius_m)
    |   movel([0.209150, -1.330470, -2.605595, -0.776324, 1.570796, 1.779946],accel_mss,speed_ms,0,blend_radius_m)
    |   movel([0.204770, -1.339489, -2.599806, -0.773094, 1.570796, 1.775566],accel_mss,speed_ms,0,blend_radius_m)
    |   movel([0.203612, -1.341935, -2.598217, -0.772237, 1.570796, 1.774408],accel_mss,speed_ms,0,blend_radius_m)
    |   movel([0.201122, -1.346997, -2.594902, -0.770490, 1.570796, 1.771918],accel_mss,speed_ms,0,blend_radius_m)
    |   movel([0.198958, -1.350636, -2.592497, -0.769256, 1.570796, 1.769754],accel_mss,speed_ms,0,blend_radius_m)
    |   movel([0.195947, -1.355258, -2.589416, -0.767715, 1.570796, 1.766744],accel_mss,speed_ms,0,blend_radius_m)
    |   movel([0.192569, -1.360174, -2.586106, -0.766108, 1.570796, 1.763365],accel_mss,speed_ms,0,blend_radius_m)
    |   movel([0.189208, -1.364803, -2.582959, -0.764627, 1.570796, 1.760004],accel_mss,speed_ms,0,blend_radius_m)
    |   movel([0.184514, -1.370947, -2.578735, -0.762707, 1.570796, 1.755310],accel_mss,speed_ms,0,blend_radius_m)
    |   movel([0.179704, -1.376969, -2.574542, -0.760878, 1.570796, 1.750501],accel_mss,speed_ms,0,blend_radius_m)
    |   movel([0.175379, -1.382092, -2.570935, -0.759362, 1.570796, 1.746175],accel_mss,speed_ms,0,blend_radius_m)
    |   movel([0.170891, -1.387072, -2.567392, -0.757925, 1.570796, 1.741687],accel_mss,speed_ms,0,blend_radius_m)
    |   movel([0.166691, -1.391423, -2.564267, -0.756699, 1.570796, 1.737488],accel_mss,speed_ms,0,blend_radius_m)
    |   movel([0.162340, -1.395619, -2.561227, -0.755543, 1.570796, 1.733136],accel_mss,speed_ms,0,blend_radius_m)
    |   movel([0.158072, -1.399425, -2.558448, -0.754516, 1.570796, 1.728868],accel_mss,speed_ms,0,blend_radius_m)
    |   movel([0.153661, -1.403041, -2.555788, -0.753560, 1.570796, 1.724458],accel_mss,speed_ms,0,blend_radius_m)
    |   movel([0.151789, -1.404490, -2.554716, -0.753182, 1.570796, 1.722585],accel_mss,speed_ms,0,blend_radius_m)
    |   movel([0.149020, -1.406449, -2.553263, -0.752677, 1.570796, 1.719817],accel_mss,speed_ms,0,blend_radius_m)
    |   movel([0.147355, -1.407509, -2.552474, -0.752406, 1.570796, 1.718151],accel_mss,speed_ms,0,blend_radius_m)
    |   movel([0.145053, -1.408865, -2.551463, -0.752061, 1.570796, 1.715849],accel_mss,speed_ms,0,blend_radius_m)
    |   movel([0.143313, -1.409705, -2.550835, -0.751849, 1.570796, 1.714109],accel_mss,speed_ms,0,blend_radius_m)
    |   movel([0.141949, -1.410128, -2.550518, -0.751743, 1.570796, 1.712745],accel_mss,speed_ms,0,blend_radius_m)
    |   movel([0.141377, -1.410203, -2.550462, -0.751724, 1.570796, 1.712173],accel_mss,speed_ms,0,blend_radius_m)
    |   movel([0.140844, -1.410179, -2.550480, -0.751730, 1.570796, 1.711641],accel_mss,speed_ms,0,blend_radius_m)
    |   movel([0.140473, -1.410059, -2.550570, -0.751760, 1.570796, 1.711269],accel_mss,speed_ms,0,blend_radius_m)
    |   movel([0.140351, -1.409839, -2.550735, -0.751816, 1.570796, 1.711148],accel_mss,speed_ms,0,blend_radius_m)
    |   movel([0.140452, -1.409431, -2.551040, -0.751918, 1.570796, 1.711248],accel_mss,speed_ms,0,blend_radius_m)
    |   movel([0.141282, -1.407598, -2.552408, -0.752383, 1.570796, 1.712079],accel_mss,speed_ms,0,blend_radius_m)
    |   movel([0.141396, -1.407144, -2.552746, -0.752499, 1.570796, 1.712192],accel_mss,speed_ms,0,blend_radius_m)
    |   movel([0.141559, -1.405710, -2.553812, -0.752867, 1.570796, 1.712356],accel_mss,speed_ms,0,blend_radius_m)
    |   movel([0.140567, -1.405019, -2.554325, -0.753046, 1.570796, 1.711363],accel_mss,speed_ms,0,blend_radius_m)
    |   movel([0.139867, -1.404428, -2.554763, -0.753199, 1.570796, 1.710663],accel_mss,speed_ms,0,blend_radius_m)
    |   movel([0.139518, -1.403860, -2.555183, -0.753346, 1.570796, 1.710314],accel_mss,speed_ms,0,blend_radius_m)
    |   movel([0.139448, -1.403163, -2.555698, -0.753528, 1.570796, 1.710244],accel_mss,speed_ms,0,blend_radius_m)
    |   movel([0.139621, -1.402183, -2.556421, -0.753785, 1.570796, 1.710418],accel_mss,speed_ms,0,blend_radius_m)
    |   movel([0.140248, -1.400511, -2.557651, -0.754227, 1.570796, 1.711044],accel_mss,speed_ms,0,blend_radius_m)
    |   movel([0.141833, -1.397393, -2.559935, -0.755061, 1.570796, 1.712629],accel_mss,speed_ms,0,blend_radius_m)
    |   movel([0.143652, -1.394106, -2.562326, -0.755956, 1.570796, 1.714448],accel_mss,speed_ms,0,blend_radius_m)
    |   movel([0.145274, -1.391509, -2.564205, -0.756675, 1.570796, 1.716071],accel_mss,speed_ms,0,blend_radius_m)
    |   movel([0.147094, -1.388979, -2.566026, -0.757384, 1.570796, 1.717890],accel_mss,speed_ms,0,blend_radius_m)
    |   movel([0.148876, -1.386858, -2.567545, -0.757986, 1.570796, 1.719672],accel_mss,speed_ms,0,blend_radius_m)
    |   movel([0.150849, -1.384891, -2.568948, -0.758550, 1.570796, 1.721645],accel_mss,speed_ms,0,blend_radius_m)
    |   movel([0.153246, -1.382834, -2.570409, -0.759146, 1.570796, 1.724043],accel_mss,speed_ms,0,blend_radius_m)
    |   movel([0.156996, -1.379586, -2.572704, -0.760099, 1.570796, 1.727793],accel_mss,speed_ms,0,blend_radius_m)
    |   movel([0.161676, -1.375096, -2.575852, -0.761441, 1.570796, 1.732473],accel_mss,speed_ms,0,blend_radius_m)
    |   movel([0.166478, -1.370191, -2.579258, -0.762941, 1.570796, 1.737275],accel_mss,speed_ms,0,blend_radius_m)
    |   movel([0.170636, -1.365609, -2.582408, -0.764372, 1.570796, 1.741432],accel_mss,speed_ms,0,blend_radius_m)
    |   movel([0.175251, -1.360034, -2.586201, -0.766154, 1.570796, 1.746048],accel_mss,speed_ms,0,blend_radius_m)
    |   movel([0.177450, -1.357175, -2.588130, -0.767085, 1.570796, 1.748246],accel_mss,speed_ms,0,blend_radius_m)
    |   movel([0.179573, -1.354270, -2.590077, -0.768042, 1.570796, 1.750369],accel_mss,speed_ms,0,blend_radius_m)
    |   movel([0.183710, -1.348173, -2.594127, -0.770089, 1.570796, 1.754506],accel_mss,speed_ms,0,blend_radius_m)
    |   movel([0.187533, -1.341932, -2.598218, -0.772238, 1.570796, 1.758329],accel_mss,speed_ms,0,blend_radius_m)
    |   movel([0.191085, -1.335461, -2.602405, -0.774523, 1.570796, 1.761881],accel_mss,speed_ms,0,blend_radius_m)
    |   movel([0.194280, -1.328893, -2.606596, -0.776900, 1.570796, 1.765077],accel_mss,speed_ms,0,blend_radius_m)
    |   movel([0.197119, -1.322219, -2.610795, -0.779375, 1.570796, 1.767915],accel_mss,speed_ms,0,blend_radius_m)
    |   movel([0.199566, -1.315497, -2.614964, -0.781928, 1.570796, 1.770362],accel_mss,speed_ms,0,blend_radius_m)
    |   movel([0.200637, -1.312119, -2.617036, -0.783234, 1.570796, 1.771434],accel_mss,speed_ms,0,blend_radius_m)
    |   movel([0.202388, -1.305483, -2.621064, -0.785842, 1.570796, 1.773185],accel_mss,speed_ms,0,blend_radius_m)
    |   movel([0.203187, -1.301766, -2.623295, -0.787329, 1.570796, 1.773983],accel_mss,speed_ms,0,blend_radius_m)
    |   movel([0.204382, -1.294903, -2.627366, -0.790120, 1.570796, 1.775178],accel_mss,speed_ms,0,blend_radius_m)
    |   movel([0.204725, -1.291897, -2.629131, -0.791361, 1.570796, 1.775521],accel_mss,speed_ms,0,blend_radius_m)
    |   movel([0.205327, -1.284412, -2.633474, -0.794503, 1.570796, 1.776123],accel_mss,speed_ms,0,blend_radius_m)
    |   movel([0.205633, -1.282908, -2.634338, -0.795143, 1.570796, 1.776429],accel_mss,speed_ms,0,blend_radius_m)
    |   movel([0.206148, -1.281361, -2.635224, -0.795804, 1.570796, 1.776944],accel_mss,speed_ms,0,blend_radius_m)
    |   movel([0.206826, -1.279924, -2.636044, -0.796421, 1.570796, 1.777623],accel_mss,speed_ms,0,blend_radius_m)
    |   movel([0.207726, -1.278501, -2.636853, -0.797034, 1.570796, 1.778522],accel_mss,speed_ms,0,blend_radius_m)
    |   movel([0.208669, -1.277360, -2.637501, -0.797528, 1.570796, 1.779466],accel_mss,speed_ms,0,blend_radius_m)
    |   movel([0.209771, -1.276327, -2.638085, -0.797977, 1.570796, 1.780568],accel_mss,speed_ms,0,blend_radius_m)
    |   movel([0.210833, -1.275621, -2.638484, -0.798284, 1.570796, 1.781629],accel_mss,speed_ms,0,blend_radius_m)
    |   movel([0.211939, -1.275197, -2.638724, -0.798469, 1.570796, 1.782735],accel_mss,speed_ms,0,blend_radius_m)
    |   movel([0.213300, -1.275053, -2.638805, -0.798531, 1.570796, 1.784096],accel_mss,speed_ms,0,blend_radius_m)
    |   movel([0.214451, -1.275318, -2.638655, -0.798416, 1.570796, 1.785247],accel_mss,speed_ms,0,blend_radius_m)
    |   movel([0.215889, -1.276097, -2.638215, -0.798076, 1.570796, 1.786685],accel_mss,speed_ms,0,blend_radius_m)
    |   movel([0.217166, -1.277055, -2.637674, -0.797661, 1.570796, 1.787963],accel_mss,speed_ms,0,blend_radius_m)
    |   movel([0.218455, -1.278351, -2.636938, -0.797099, 1.570796, 1.789252],accel_mss,speed_ms,0,blend_radius_m)
    |   movel([0.219548, -1.279817, -2.636105, -0.796467, 1.570796, 1.790344],accel_mss,speed_ms,0,blend_radius_m)
    |   movel([0.220437, -1.281441, -2.635178, -0.795770, 1.570796, 1.791233],accel_mss,speed_ms,0,blend_radius_m)
    |   movel([0.221118, -1.283205, -2.634167, -0.795017, 1.570796, 1.791914],accel_mss,speed_ms,0,blend_radius_m)
    |   movel([0.221734, -1.285674, -2.632746, -0.793968, 1.570796, 1.792530],accel_mss,speed_ms,0,blend_radius_m)
    |   movel([0.222086, -1.288290, -2.631232, -0.792867, 1.570796, 1.792882],accel_mss,speed_ms,0,blend_radius_m)
    |   movel([0.222237, -1.291669, -2.629264, -0.791456, 1.570796, 1.793033],accel_mss,speed_ms,0,blend_radius_m)
    |   movel([0.222220, -1.301708, -2.623329, -0.787352, 1.570796, 1.793016],accel_mss,speed_ms,0,blend_radius_m)
    |   movel([0.222375, -1.305332, -2.621155, -0.785902, 1.570796, 1.793171],accel_mss,speed_ms,0,blend_radius_m)
    |   movel([0.222701, -1.308078, -2.619495, -0.784815, 1.570796, 1.793498],accel_mss,speed_ms,0,blend_radius_m)
    |   movel([0.223235, -1.310268, -2.618166, -0.783956, 1.570796, 1.794031],accel_mss,speed_ms,0,blend_radius_m)
    |   movel([0.224029, -1.312156, -2.617014, -0.783220, 1.570796, 1.794826],accel_mss,speed_ms,0,blend_radius_m)
    |   movel([0.224382, -1.312554, -2.616770, -0.783065, 1.570796, 1.795178],accel_mss,speed_ms,0,blend_radius_m)
    |   movel([0.224907, -1.312768, -2.616639, -0.782982, 1.570796, 1.795704],accel_mss,speed_ms,0,blend_radius_m)
    |   movel([0.225531, -1.312759, -2.616645, -0.782985, 1.570796, 1.796327],accel_mss,speed_ms,0,blend_radius_m)
    |   movel([0.226215, -1.312532, -2.616783, -0.783073, 1.570796, 1.797011],accel_mss,speed_ms,0,blend_radius_m)
    |   movel([0.228551, -1.311256, -2.617563, -0.783570, 1.570796, 1.799347],accel_mss,speed_ms,0,blend_radius_m)
    |   movel([0.230258, -1.310138, -2.618245, -0.784007, 1.570796, 1.801054],accel_mss,speed_ms,0,blend_radius_m)
    |   movel([0.232043, -1.308830, -2.619039, -0.784519, 1.570796, 1.802839],accel_mss,speed_ms,0,blend_radius_m)
    |   movel([0.237010, -1.304758, -2.621500, -0.786131, 1.570796, 1.807806],accel_mss,speed_ms,0,blend_radius_m)
    |   movel([0.241343, -1.301159, -2.623657, -0.787573, 1.570796, 1.812139],accel_mss,speed_ms,0,blend_radius_m)
    |   movel([0.244377, -1.298858, -2.625027, -0.788504, 1.570796, 1.815173],accel_mss,speed_ms,0,blend_radius_m)
    |   movel([0.246680, -1.297398, -2.625893, -0.789098, 1.570796, 1.817476],accel_mss,speed_ms,0,blend_radius_m)
    |   movel([0.247621, -1.296933, -2.626168, -0.789288, 1.570796, 1.818417],accel_mss,speed_ms,0,blend_radius_m)
    |   movel([0.248567, -1.296585, -2.626374, -0.789430, 1.570796, 1.819363],accel_mss,speed_ms,0,blend_radius_m)
    |   movel([0.249533, -1.296414, -2.626475, -0.789500, 1.570796, 1.820329],accel_mss,speed_ms,0,blend_radius_m)
    |   movel([0.250363, -1.296501, -2.626423, -0.789464, 1.570796, 1.821159],accel_mss,speed_ms,0,blend_radius_m)
    |   movel([0.250994, -1.296850, -2.626217, -0.789322, 1.570796, 1.821790],accel_mss,speed_ms,0,blend_radius_m)
    |   movel([0.251387, -1.297428, -2.625875, -0.789086, 1.570796, 1.822183],accel_mss,speed_ms,0,blend_radius_m)
    |   movel([0.251614, -1.298257, -2.625384, -0.788748, 1.570796, 1.822410],accel_mss,speed_ms,0,blend_radius_m)
    |   movel([0.251693, -1.299162, -2.624847, -0.788381, 1.570796, 1.822489],accel_mss,speed_ms,0,blend_radius_m)
    |   movel([0.251483, -1.301470, -2.623471, -0.787448, 1.570796, 1.822279],accel_mss,speed_ms,0,blend_radius_m)
    |   movel([0.250799, -1.304176, -2.621850, -0.786363, 1.570796, 1.821595],accel_mss,speed_ms,0,blend_radius_m)
    |   movel([0.249676, -1.307108, -2.620083, -0.785198, 1.570796, 1.820473],accel_mss,speed_ms,0,blend_radius_m)
    |   movel([0.248671, -1.309163, -2.618837, -0.784389, 1.570796, 1.819468],accel_mss,speed_ms,0,blend_radius_m)
    |   movel([0.248375, -1.309664, -2.618533, -0.784192, 1.570796, 1.819172],accel_mss,speed_ms,0,blend_radius_m)
    |   speed_ms = 0.005
    |   movel([0.248375, -1.300507, -2.614217, -0.797665, 1.570796, 1.819172],accel_mss,speed_ms,0,blend_radius_m)
    |   speed_ms = 0.040
    |   movel([0.250519, -1.290806, -2.619977, -0.801606, 1.570796, 1.821316],accel_mss,speed_ms,0,blend_radius_m)
    |   speed_ms = 0.005
    |   movel([0.250519, -1.300019, -2.624337, -0.788033, 1.570796, 1.821316],accel_mss,speed_ms,0,blend_radius_m)
    |   speed_ms = 0.025
    |   movel([0.250460, -1.300588, -2.623997, -0.787803, 1.570796, 1.821256],accel_mss,speed_ms,0,blend_radius_m)
    |   movel([0.249846, -1.303470, -2.622274, -0.786645, 1.570796, 1.820642],accel_mss,speed_ms,0,blend_radius_m)
    |   movel([0.249048, -1.306052, -2.620721, -0.785617, 1.570796, 1.819844],accel_mss,speed_ms,0,blend_radius_m)
    |   movel([0.248096, -1.308280, -2.619373, -0.784736, 1.570796, 1.818892],accel_mss,speed_ms,0,blend_radius_m)
    |   movel([0.246813, -1.310542, -2.617999, -0.783849, 1.570796, 1.817609],accel_mss,speed_ms,0,blend_radius_m)
    |   movel([0.244994, -1.313225, -2.616360, -0.782805, 1.570796, 1.815791],accel_mss,speed_ms,0,blend_radius_m)
    |   movel([0.242792, -1.316032, -2.614634, -0.781723, 1.570796, 1.813588],accel_mss,speed_ms,0,blend_radius_m)
    |   movel([0.240292, -1.318750, -2.612954, -0.780685, 1.570796, 1.811088],accel_mss,speed_ms,0,blend_radius_m)
    |   movel([0.237114, -1.321776, -2.611071, -0.779541, 1.570796, 1.807910],accel_mss,speed_ms,0,blend_radius_m)
    |   movel([0.232770, -1.325581, -2.608687, -0.778121, 1.570796, 1.803567],accel_mss,speed_ms,0,blend_radius_m)
    |   movel([0.227732, -1.329732, -2.606064, -0.776593, 1.570796, 1.798529],accel_mss,speed_ms,0,blend_radius_m)
    |   movel([0.225835, -1.331172, -2.605149, -0.776069, 1.570796, 1.796631],accel_mss,speed_ms,0,blend_radius_m)
    |   movel([0.223885, -1.332518, -2.604290, -0.775581, 1.570796, 1.794681],accel_mss,speed_ms,0,blend_radius_m)
    |   movel([0.222342, -1.333460, -2.603688, -0.775241, 1.570796, 1.793138],accel_mss,speed_ms,0,blend_radius_m)
    |   movel([0.220770, -1.334287, -2.603158, -0.774943, 1.570796, 1.791566],accel_mss,speed_ms,0,blend_radius_m)
    |   movel([0.219422, -1.334850, -2.602798, -0.774742, 1.570796, 1.790218],accel_mss,speed_ms,0,blend_radius_m)
    |   movel([0.218086, -1.335223, -2.602558, -0.774608, 1.570796, 1.788882],accel_mss,speed_ms,0,blend_radius_m)
    |   movel([0.217116, -1.335369, -2.602464, -0.774556, 1.570796, 1.787912],accel_mss,speed_ms,0,blend_radius_m)
    |   movel([0.216193, -1.335388, -2.602452, -0.774549, 1.570796, 1.786989],accel_mss,speed_ms,0,blend_radius_m)
    |   movel([0.215429, -1.335268, -2.602529, -0.774592, 1.570796, 1.786226],accel_mss,speed_ms,0,blend_radius_m)
    |   movel([0.214773, -1.334995, -2.602704, -0.774690, 1.570796, 1.785569],accel_mss,speed_ms,0,blend_radius_m)
    |   movel([0.214128, -1.334524, -2.603007, -0.774859, 1.570796, 1.784924],accel_mss,speed_ms,0,blend_radius_m)
    |   movel([0.213612, -1.333932, -2.603386, -0.775071, 1.570796, 1.784409],accel_mss,speed_ms,0,blend_radius_m)
    |   movel([0.211817, -1.330718, -2.605437, -0.776234, 1.570796, 1.782614],accel_mss,speed_ms,0,blend_radius_m)
    |   movel([0.211115, -1.329702, -2.606083, -0.776604, 1.570796, 1.781911],accel_mss,speed_ms,0,blend_radius_m)
    |   movel([0.210448, -1.328985, -2.606538, -0.776867, 1.570796, 1.781244],accel_mss,speed_ms,0,blend_radius_m)
    |   movel([0.209929, -1.328794, -2.606659, -0.776936, 1.570796, 1.780726],accel_mss,speed_ms,0,blend_radius_m)
    |   movel([0.209450, -1.328951, -2.606559, -0.776879, 1.570796, 1.780246],accel_mss,speed_ms,0,blend_radius_m)
    |   movel([0.208919, -1.329408, -2.606270, -0.776712, 1.570796, 1.779716],accel_mss,speed_ms,0,blend_radius_m)
    |   movel([0.208337, -1.330187, -2.605775, -0.776427, 1.570796, 1.779133],accel_mss,speed_ms,0,blend_radius_m)
    |   movel([0.207698, -1.331307, -2.605062, -0.776020, 1.570796, 1.778494],accel_mss,speed_ms,0,blend_radius_m)
    |   movel([0.203802, -1.339400, -2.599864, -0.773125, 1.570796, 1.774598],accel_mss,speed_ms,0,blend_radius_m)
    |   movel([0.201051, -1.345101, -2.596148, -0.771140, 1.570796, 1.771847],accel_mss,speed_ms,0,blend_radius_m)
    |   movel([0.199031, -1.348896, -2.593649, -0.769844, 1.570796, 1.769827],accel_mss,speed_ms,0,blend_radius_m)
    |   movel([0.196849, -1.352451, -2.591291, -0.768647, 1.570796, 1.767645],accel_mss,speed_ms,0,blend_radius_m)
    |   movel([0.193643, -1.357203, -2.588111, -0.767075, 1.570796, 1.764439],accel_mss,speed_ms,0,blend_radius_m)
    |   movel([0.190757, -1.361295, -2.585347, -0.765747, 1.570796, 1.761553],accel_mss,speed_ms,0,blend_radius_m)
    |   movel([0.184674, -1.369428, -2.579784, -0.763177, 1.570796, 1.755470],accel_mss,speed_ms,0,blend_radius_m)
    |   movel([0.181495, -1.373463, -2.576989, -0.761936, 1.570796, 1.752291],accel_mss,speed_ms,0,blend_radius_m)
    |   movel([0.175156, -1.381102, -2.571635, -0.759652, 1.570796, 1.745953],accel_mss,speed_ms,0,blend_radius_m)
    |   movel([0.172202, -1.384466, -2.569250, -0.758672, 1.570796, 1.742998],accel_mss,speed_ms,0,blend_radius_m)
    |   movel([0.169173, -1.387760, -2.566900, -0.757729, 1.570796, 1.739969],accel_mss,speed_ms,0,blend_radius_m)
    |   movel([0.165913, -1.391121, -2.564485, -0.756783, 1.570796, 1.736709],accel_mss,speed_ms,0,blend_radius_m)
    |   movel([0.162557, -1.394381, -2.562127, -0.755881, 1.570796, 1.733354],accel_mss,speed_ms,0,blend_radius_m)
    |   movel([0.159209, -1.397439, -2.559901, -0.755049, 1.570796, 1.730005],accel_mss,speed_ms,0,blend_radius_m)
    |   movel([0.155768, -1.400382, -2.557746, -0.754261, 1.570796, 1.726564],accel_mss,speed_ms,0,blend_radius_m)
    |   movel([0.152646, -1.402878, -2.555908, -0.753603, 1.570796, 1.723443],accel_mss,speed_ms,0,blend_radius_m)
    |   movel([0.149447, -1.405257, -2.554148, -0.752984, 1.570796, 1.720243],accel_mss,speed_ms,0,blend_radius_m)
    |   movel([0.146921, -1.406922, -2.552912, -0.752556, 1.570796, 1.717718],accel_mss,speed_ms,0,blend_radius_m)
    |   movel([0.144306, -1.408362, -2.551839, -0.752189, 1.570796, 1.715102],accel_mss,speed_ms,0,blend_radius_m)
    |   movel([0.143331, -1.408808, -2.551505, -0.752076, 1.570796, 1.714128],accel_mss,speed_ms,0,blend_radius_m)
    |   movel([0.141724, -1.409323, -2.551121, -0.751946, 1.570796, 1.712520],accel_mss,speed_ms,0,blend_radius_m)
    |   movel([0.141584, -1.409215, -2.551201, -0.751973, 1.570796, 1.712380],accel_mss,speed_ms,0,blend_radius_m)
    |   movel([0.142049, -1.407986, -2.552119, -0.752284, 1.570796, 1.712845],accel_mss,speed_ms,0,blend_radius_m)
    |   movel([0.142441, -1.406680, -2.553091, -0.752618, 1.570796, 1.713238],accel_mss,speed_ms,0,blend_radius_m)
    |   movel([0.142466, -1.405609, -2.553887, -0.752893, 1.570796, 1.713262],accel_mss,speed_ms,0,blend_radius_m)
    |   movel([0.142107, -1.404779, -2.554502, -0.753108, 1.570796, 1.712903],accel_mss,speed_ms,0,blend_radius_m)
    |   movel([0.140998, -1.403900, -2.555153, -0.753336, 1.570796, 1.711794],accel_mss,speed_ms,0,blend_radius_m)
